(* Logix 5000 project; controller reports 1756-L63 rev 20.11; software revision 20.04; part 24 of 52 *)

        [1606].log_data[4].valid := 1, [1606].log_data[5].valid := 1, [1606].log_data[6].valid := 1, [1606].log_data[7].valid := 1, [1606].log_data[8].valid := 1, [1606].log_data[9].valid := 1, [1606].log_data[10].valid := 1, [1606].log_data[11].valid := 1, [1606].log_data[12].valid := 1, [1606].log_data[13].valid := 1, [1606].log_data[14].valid := 1, [1606].log_data[15].valid := 1, [1606].log_data[16].valid := 1, [1606].log_data[17].valid := 1, [1606].log_data[18].valid := 1, [1606].log_data[19].valid := 1, [1606].time.Year := 2023, [1606].time.Month := 1, [1606].time.Day := 15, [1606].time.Hour := 6, [1606].time.Minute := 14, [1606].time.Second := 59, [1607].log_data[0].min := 1.0, [1607].log_data[0].max := 1.0, [1607].log_data[0].total := 300.0, [1607].log_data[0].time := 300.0, [1607].log_data[0].minminute := 15, [1607].log_data[0].maxminute := 15, [1607].log_data[0].valid := 1, [1607].log_data[1].valid := 1, [1607].log_data[2].valid := 1, [1607].log_data[3].valid := 1, [1607].log_data[4].valid := 1, [1607].log_data[5].valid := 1, [1607].log_data[6].valid := 1, [1607].log_data[7].valid := 1, [1607].log_data[8].valid := 1, [1607].log_data[9].valid := 1, [1607].log_data[10].valid := 1, [1607].log_data[11].valid := 1, [1607].log_data[12].valid := 1, [1607].log_data[13].valid := 1, [1607].log_data[14].valid := 1, [1607].log_data[15].valid := 1, [1607].log_data[16].valid := 1, [1607].log_data[17].valid := 1, [1607].log_data[18].valid := 1, [1607].log_data[19].valid := 1, [1607].time.Year := 2023, [1607].time.Month := 1, [1607].time.Day := 15, [1607].time.Hour := 6, [1607].time.Minute := 19, [1607].time.Second := 59, [1608].log_data[0].min := 1.0, [1608].log_data[0].max := 1.0, [1608].log_data[0].total := 300.0, [1608].log_data[0].time := 300.0, [1608].log_data[0].minminute := 20, [1608].log_data[0].maxminute := 20,
        [1608].log_data[0].valid := 1, [1608].log_data[1].valid := 1, [1608].log_data[2].valid := 1, [1608].log_data[3].valid := 1, [1608].log_data[4].valid := 1, [1608].log_data[5].valid := 1, [1608].log_data[6].valid := 1, [1608].log_data[7].valid := 1, [1608].log_data[8].valid := 1, [1608].log_data[9].valid := 1, [1608].log_data[10].valid := 1, [1608].log_data[11].valid := 1, [1608].log_data[12].valid := 1, [1608].log_data[13].valid := 1, [1608].log_data[14].valid := 1, [1608].log_data[15].valid := 1, [1608].log_data[16].valid := 1, [1608].log_data[17].valid := 1, [1608].log_data[18].valid := 1, [1608].log_data[19].valid := 1, [1608].time.Year := 2023, [1608].time.Month := 1, [1608].time.Day := 15, [1608].time.Hour := 6, [1608].time.Minute := 24, [1608].time.Second := 59, [1609].log_data[0].min := 1.0, [1609].log_data[0].max := 1.0, [1609].log_data[0].total := 300.0, [1609].log_data[0].time := 300.0, [1609].log_data[0].minminute := 25, [1609].log_data[0].maxminute := 25, [1609].log_data[0].valid := 1, [1609].log_data[1].valid := 1, [1609].log_data[2].valid := 1, [1609].log_data[3].valid := 1, [1609].log_data[4].valid := 1, [1609].log_data[5].valid := 1, [1609].log_data[6].valid := 1, [1609].log_data[7].valid := 1, [1609].log_data[8].valid := 1, [1609].log_data[9].valid := 1, [1609].log_data[10].valid := 1, [1609].log_data[11].valid := 1, [1609].log_data[12].valid := 1, [1609].log_data[13].valid := 1, [1609].log_data[14].valid := 1, [1609].log_data[15].valid := 1, [1609].log_data[16].valid := 1, [1609].log_data[17].valid := 1, [1609].log_data[18].valid := 1, [1609].log_data[19].valid := 1, [1609].time.Year := 2023, [1609].time.Month := 1, [1609].time.Day := 15, [1609].time.Hour := 6, [1609].time.Minute := 29, [1609].time.Second := 59, [1610].log_data[0].min := 1.0, [1610].log_data[0].max := 1.0,
        [1610].log_data[0].total := 300.0, [1610].log_data[0].time := 300.0, [1610].log_data[0].minminute := 30, [1610].log_data[0].maxminute := 30, [1610].log_data[0].valid := 1, [1610].log_data[1].valid := 1, [1610].log_data[2].valid := 1, [1610].log_data[3].valid := 1, [1610].log_data[4].valid := 1, [1610].log_data[5].valid := 1, [1610].log_data[6].valid := 1, [1610].log_data[7].valid := 1, [1610].log_data[8].valid := 1, [1610].log_data[9].valid := 1, [1610].log_data[10].valid := 1, [1610].log_data[11].valid := 1, [1610].log_data[12].valid := 1, [1610].log_data[13].valid := 1, [1610].log_data[14].valid := 1, [1610].log_data[15].valid := 1, [1610].log_data[16].valid := 1, [1610].log_data[17].valid := 1, [1610].log_data[18].valid := 1, [1610].log_data[19].valid := 1, [1610].time.Year := 2023, [1610].time.Month := 1, [1610].time.Day := 15, [1610].time.Hour := 6, [1610].time.Minute := 34, [1610].time.Second := 59, [1611].log_data[0].min := 1.0, [1611].log_data[0].max := 1.0, [1611].log_data[0].total := 300.0, [1611].log_data[0].time := 300.0, [1611].log_data[0].minminute := 35, [1611].log_data[0].maxminute := 35, [1611].log_data[0].valid := 1, [1611].log_data[1].valid := 1, [1611].log_data[2].valid := 1, [1611].log_data[3].valid := 1, [1611].log_data[4].valid := 1, [1611].log_data[5].valid := 1, [1611].log_data[6].valid := 1, [1611].log_data[7].valid := 1, [1611].log_data[8].valid := 1, [1611].log_data[9].valid := 1, [1611].log_data[10].valid := 1, [1611].log_data[11].valid := 1, [1611].log_data[12].valid := 1, [1611].log_data[13].valid := 1, [1611].log_data[14].valid := 1, [1611].log_data[15].valid := 1, [1611].log_data[16].valid := 1, [1611].log_data[17].valid := 1, [1611].log_data[18].valid := 1, [1611].log_data[19].valid := 1, [1611].time.Year := 2023, [1611].time.Month := 1, [1611].time.Day := 15, [1611].time.Hour := 6,
        [1611].time.Minute := 39, [1611].time.Second := 59, [1612].log_data[0].min := 1.0, [1612].log_data[0].max := 1.0, [1612].log_data[0].total := 300.0, [1612].log_data[0].time := 300.0, [1612].log_data[0].minminute := 40, [1612].log_data[0].maxminute := 40, [1612].log_data[0].valid := 1, [1612].log_data[1].valid := 1, [1612].log_data[2].valid := 1, [1612].log_data[3].valid := 1, [1612].log_data[4].valid := 1, [1612].log_data[5].valid := 1, [1612].log_data[6].valid := 1, [1612].log_data[7].valid := 1, [1612].log_data[8].valid := 1, [1612].log_data[9].valid := 1, [1612].log_data[10].valid := 1, [1612].log_data[11].valid := 1, [1612].log_data[12].valid := 1, [1612].log_data[13].valid := 1, [1612].log_data[14].valid := 1, [1612].log_data[15].valid := 1, [1612].log_data[16].valid := 1, [1612].log_data[17].valid := 1, [1612].log_data[18].valid := 1, [1612].log_data[19].valid := 1, [1612].time.Year := 2023, [1612].time.Month := 1, [1612].time.Day := 15, [1612].time.Hour := 6, [1612].time.Minute := 44, [1612].time.Second := 59, [1613].log_data[0].min := 1.0, [1613].log_data[0].max := 1.0, [1613].log_data[0].total := 300.0, [1613].log_data[0].time := 300.0, [1613].log_data[0].minminute := 45, [1613].log_data[0].maxminute := 45, [1613].log_data[0].valid := 1, [1613].log_data[1].valid := 1, [1613].log_data[2].valid := 1, [1613].log_data[3].valid := 1, [1613].log_data[4].valid := 1, [1613].log_data[5].valid := 1, [1613].log_data[6].valid := 1, [1613].log_data[7].valid := 1, [1613].log_data[8].valid := 1, [1613].log_data[9].valid := 1, [1613].log_data[10].valid := 1, [1613].log_data[11].valid := 1, [1613].log_data[12].valid := 1, [1613].log_data[13].valid := 1, [1613].log_data[14].valid := 1, [1613].log_data[15].valid := 1, [1613].log_data[16].valid := 1, [1613].log_data[17].valid := 1, [1613].log_data[18].valid := 1, [1613].log_data[19].valid := 1,
        [1613].time.Year := 2023, [1613].time.Month := 1, [1613].time.Day := 15, [1613].time.Hour := 6, [1613].time.Minute := 49, [1613].time.Second := 59, [1614].log_data[0].min := 1.0, [1614].log_data[0].max := 1.0, [1614].log_data[0].total := 300.0, [1614].log_data[0].time := 300.0, [1614].log_data[0].minminute := 50, [1614].log_data[0].maxminute := 50, [1614].log_data[0].valid := 1, [1614].log_data[1].valid := 1, [1614].log_data[2].valid := 1, [1614].log_data[3].valid := 1, [1614].log_data[4].valid := 1, [1614].log_data[5].valid := 1, [1614].log_data[6].valid := 1, [1614].log_data[7].valid := 1, [1614].log_data[8].valid := 1, [1614].log_data[9].valid := 1, [1614].log_data[10].valid := 1, [1614].log_data[11].valid := 1, [1614].log_data[12].valid := 1, [1614].log_data[13].valid := 1, [1614].log_data[14].valid := 1, [1614].log_data[15].valid := 1, [1614].log_data[16].valid := 1, [1614].log_data[17].valid := 1, [1614].log_data[18].valid := 1, [1614].log_data[19].valid := 1, [1614].time.Year := 2023, [1614].time.Month := 1, [1614].time.Day := 15, [1614].time.Hour := 6, [1614].time.Minute := 54, [1614].time.Second := 59, [1615].log_data[0].min := 1.0, [1615].log_data[0].max := 1.0, [1615].log_data[0].total := 300.0, [1615].log_data[0].time := 300.0, [1615].log_data[0].minminute := 55, [1615].log_data[0].maxminute := 55, [1615].log_data[0].valid := 1, [1615].log_data[1].valid := 1, [1615].log_data[2].valid := 1, [1615].log_data[3].valid := 1, [1615].log_data[4].valid := 1, [1615].log_data[5].valid := 1, [1615].log_data[6].valid := 1, [1615].log_data[7].valid := 1, [1615].log_data[8].valid := 1, [1615].log_data[9].valid := 1, [1615].log_data[10].valid := 1, [1615].log_data[11].valid := 1, [1615].log_data[12].valid := 1, [1615].log_data[13].valid := 1, [1615].log_data[14].valid := 1, [1615].log_data[15].valid := 1,
        [1615].log_data[16].valid := 1, [1615].log_data[17].valid := 1, [1615].log_data[18].valid := 1, [1615].log_data[19].valid := 1, [1615].time.Year := 2023, [1615].time.Month := 1, [1615].time.Day := 15, [1615].time.Hour := 6, [1615].time.Minute := 59, [1615].time.Second := 59, [1616].log_data[0].min := 1.0, [1616].log_data[0].max := 1.0, [1616].log_data[0].total := 300.0, [1616].log_data[0].time := 300.0, [1616].log_data[0].valid := 1, [1616].log_data[1].valid := 1, [1616].log_data[2].valid := 1, [1616].log_data[3].valid := 1, [1616].log_data[4].valid := 1, [1616].log_data[5].valid := 1, [1616].log_data[6].valid := 1, [1616].log_data[7].valid := 1, [1616].log_data[8].valid := 1, [1616].log_data[9].valid := 1, [1616].log_data[10].valid := 1, [1616].log_data[11].valid := 1, [1616].log_data[12].valid := 1, [1616].log_data[13].valid := 1, [1616].log_data[14].valid := 1, [1616].log_data[15].valid := 1, [1616].log_data[16].valid := 1, [1616].log_data[17].valid := 1, [1616].log_data[18].valid := 1, [1616].log_data[19].valid := 1, [1616].time.Year := 2023, [1616].time.Month := 1, [1616].time.Day := 15, [1616].time.Hour := 7, [1616].time.Minute := 4, [1616].time.Second := 59, [1617].log_data[0].min := 1.0, [1617].log_data[0].max := 1.0, [1617].log_data[0].total := 300.0, [1617].log_data[0].time := 300.0, [1617].log_data[0].minminute := 5, [1617].log_data[0].maxminute := 5, [1617].log_data[0].valid := 1, [1617].log_data[1].valid := 1, [1617].log_data[2].valid := 1, [1617].log_data[3].valid := 1, [1617].log_data[4].valid := 1, [1617].log_data[5].valid := 1, [1617].log_data[6].valid := 1, [1617].log_data[7].valid := 1, [1617].log_data[8].valid := 1, [1617].log_data[9].valid := 1, [1617].log_data[10].valid := 1, [1617].log_data[11].valid := 1, [1617].log_data[12].valid := 1, [1617].log_data[13].valid := 1,
        [1617].log_data[14].valid := 1, [1617].log_data[15].valid := 1, [1617].log_data[16].valid := 1, [1617].log_data[17].valid := 1, [1617].log_data[18].valid := 1, [1617].log_data[19].valid := 1, [1617].time.Year := 2023, [1617].time.Month := 1, [1617].time.Day := 15, [1617].time.Hour := 7, [1617].time.Minute := 9, [1617].time.Second := 59, [1618].log_data[0].min := 1.0, [1618].log_data[0].max := 1.0, [1618].log_data[0].total := 300.0, [1618].log_data[0].time := 300.0, [1618].log_data[0].minminute := 10, [1618].log_data[0].maxminute := 10, [1618].log_data[0].valid := 1, [1618].log_data[1].valid := 1, [1618].log_data[2].valid := 1, [1618].log_data[3].valid := 1, [1618].log_data[4].valid := 1, [1618].log_data[5].valid := 1, [1618].log_data[6].valid := 1, [1618].log_data[7].valid := 1, [1618].log_data[8].valid := 1, [1618].log_data[9].valid := 1, [1618].log_data[10].valid := 1, [1618].log_data[11].valid := 1, [1618].log_data[12].valid := 1, [1618].log_data[13].valid := 1, [1618].log_data[14].valid := 1, [1618].log_data[15].valid := 1, [1618].log_data[16].valid := 1, [1618].log_data[17].valid := 1, [1618].log_data[18].valid := 1, [1618].log_data[19].valid := 1, [1618].time.Year := 2023, [1618].time.Month := 1, [1618].time.Day := 15, [1618].time.Hour := 7, [1618].time.Minute := 14, [1618].time.Second := 59, [1619].log_data[0].min := 1.0, [1619].log_data[0].max := 1.0, [1619].log_data[0].total := 300.0, [1619].log_data[0].time := 300.0, [1619].log_data[0].minminute := 15, [1619].log_data[0].maxminute := 15, [1619].log_data[0].valid := 1, [1619].log_data[1].valid := 1, [1619].log_data[2].valid := 1, [1619].log_data[3].valid := 1, [1619].log_data[4].valid := 1, [1619].log_data[5].valid := 1, [1619].log_data[6].valid := 1, [1619].log_data[7].valid := 1, [1619].log_data[8].valid := 1, [1619].log_data[9].valid := 1,
        [1619].log_data[10].valid := 1, [1619].log_data[11].valid := 1, [1619].log_data[12].valid := 1, [1619].log_data[13].valid := 1, [1619].log_data[14].valid := 1, [1619].log_data[15].valid := 1, [1619].log_data[16].valid := 1, [1619].log_data[17].valid := 1, [1619].log_data[18].valid := 1, [1619].log_data[19].valid := 1, [1619].time.Year := 2023, [1619].time.Month := 1, [1619].time.Day := 15, [1619].time.Hour := 7, [1619].time.Minute := 19, [1619].time.Second := 59, [1620].log_data[0].min := 1.0, [1620].log_data[0].max := 1.0, [1620].log_data[0].total := 300.0, [1620].log_data[0].time := 300.0, [1620].log_data[0].minminute := 20, [1620].log_data[0].maxminute := 20, [1620].log_data[0].valid := 1, [1620].log_data[1].valid := 1, [1620].log_data[2].valid := 1, [1620].log_data[3].valid := 1, [1620].log_data[4].valid := 1, [1620].log_data[5].valid := 1, [1620].log_data[6].valid := 1, [1620].log_data[7].valid := 1, [1620].log_data[8].valid := 1, [1620].log_data[9].valid := 1, [1620].log_data[10].valid := 1, [1620].log_data[11].valid := 1, [1620].log_data[12].valid := 1, [1620].log_data[13].valid := 1, [1620].log_data[14].valid := 1, [1620].log_data[15].valid := 1, [1620].log_data[16].valid := 1, [1620].log_data[17].valid := 1, [1620].log_data[18].valid := 1, [1620].log_data[19].valid := 1, [1620].time.Year := 2023, [1620].time.Month := 1, [1620].time.Day := 15, [1620].time.Hour := 7, [1620].time.Minute := 24, [1620].time.Second := 59, [1621].log_data[0].min := 1.0, [1621].log_data[0].max := 1.0, [1621].log_data[0].total := 300.0, [1621].log_data[0].time := 300.0, [1621].log_data[0].minminute := 25, [1621].log_data[0].maxminute := 25, [1621].log_data[0].valid := 1, [1621].log_data[1].valid := 1, [1621].log_data[2].valid := 1, [1621].log_data[3].valid := 1, [1621].log_data[4].valid := 1, [1621].log_data[5].valid := 1,
        [1621].log_data[6].valid := 1, [1621].log_data[7].valid := 1, [1621].log_data[8].valid := 1, [1621].log_data[9].valid := 1, [1621].log_data[10].valid := 1, [1621].log_data[11].valid := 1, [1621].log_data[12].valid := 1, [1621].log_data[13].valid := 1, [1621].log_data[14].valid := 1, [1621].log_data[15].valid := 1, [1621].log_data[16].valid := 1, [1621].log_data[17].valid := 1, [1621].log_data[18].valid := 1, [1621].log_data[19].valid := 1, [1621].time.Year := 2023, [1621].time.Month := 1, [1621].time.Day := 15, [1621].time.Hour := 7, [1621].time.Minute := 29, [1621].time.Second := 59, [1622].log_data[0].min := 1.0, [1622].log_data[0].max := 1.0, [1622].log_data[0].total := 300.0, [1622].log_data[0].time := 300.0, [1622].log_data[0].minminute := 30, [1622].log_data[0].maxminute := 30, [1622].log_data[0].valid := 1, [1622].log_data[1].valid := 1, [1622].log_data[2].valid := 1, [1622].log_data[3].valid := 1, [1622].log_data[4].valid := 1, [1622].log_data[5].valid := 1, [1622].log_data[6].valid := 1, [1622].log_data[7].valid := 1, [1622].log_data[8].valid := 1, [1622].log_data[9].valid := 1, [1622].log_data[10].valid := 1, [1622].log_data[11].valid := 1, [1622].log_data[12].valid := 1, [1622].log_data[13].valid := 1, [1622].log_data[14].valid := 1, [1622].log_data[15].valid := 1, [1622].log_data[16].valid := 1, [1622].log_data[17].valid := 1, [1622].log_data[18].valid := 1, [1622].log_data[19].valid := 1, [1622].time.Year := 2023, [1622].time.Month := 1, [1622].time.Day := 15, [1622].time.Hour := 7, [1622].time.Minute := 34, [1622].time.Second := 59, [1623].log_data[0].min := 1.0, [1623].log_data[0].max := 1.0, [1623].log_data[0].total := 300.0, [1623].log_data[0].time := 300.0, [1623].log_data[0].minminute := 35, [1623].log_data[0].maxminute := 35, [1623].log_data[0].valid := 1, [1623].log_data[1].valid := 1,
        [1623].log_data[2].valid := 1, [1623].log_data[3].valid := 1, [1623].log_data[4].valid := 1, [1623].log_data[5].valid := 1, [1623].log_data[6].valid := 1, [1623].log_data[7].valid := 1, [1623].log_data[8].valid := 1, [1623].log_data[9].valid := 1, [1623].log_data[10].valid := 1, [1623].log_data[11].valid := 1, [1623].log_data[12].valid := 1, [1623].log_data[13].valid := 1, [1623].log_data[14].valid := 1, [1623].log_data[15].valid := 1, [1623].log_data[16].valid := 1, [1623].log_data[17].valid := 1, [1623].log_data[18].valid := 1, [1623].log_data[19].valid := 1, [1623].time.Year := 2023, [1623].time.Month := 1, [1623].time.Day := 15, [1623].time.Hour := 7, [1623].time.Minute := 39, [1623].time.Second := 59, [1624].log_data[0].min := 1.0, [1624].log_data[0].max := 1.0, [1624].log_data[0].total := 300.0, [1624].log_data[0].time := 300.0, [1624].log_data[0].minminute := 40, [1624].log_data[0].maxminute := 40, [1624].log_data[0].valid := 1, [1624].log_data[1].valid := 1, [1624].log_data[2].valid := 1, [1624].log_data[3].valid := 1, [1624].log_data[4].valid := 1, [1624].log_data[5].valid := 1, [1624].log_data[6].valid := 1, [1624].log_data[7].valid := 1, [1624].log_data[8].valid := 1, [1624].log_data[9].valid := 1, [1624].log_data[10].valid := 1, [1624].log_data[11].valid := 1, [1624].log_data[12].valid := 1, [1624].log_data[13].valid := 1, [1624].log_data[14].valid := 1, [1624].log_data[15].valid := 1, [1624].log_data[16].valid := 1, [1624].log_data[17].valid := 1, [1624].log_data[18].valid := 1, [1624].log_data[19].valid := 1, [1624].time.Year := 2023, [1624].time.Month := 1, [1624].time.Day := 15, [1624].time.Hour := 7, [1624].time.Minute := 44, [1624].time.Second := 59, [1625].log_data[0].min := 1.0, [1625].log_data[0].max := 1.0, [1625].log_data[0].total := 300.0, [1625].log_data[0].time := 300.0,
        [1625].log_data[0].minminute := 45, [1625].log_data[0].maxminute := 45, [1625].log_data[0].valid := 1, [1625].log_data[1].valid := 1, [1625].log_data[2].valid := 1, [1625].log_data[3].valid := 1, [1625].log_data[4].valid := 1, [1625].log_data[5].valid := 1, [1625].log_data[6].valid := 1, [1625].log_data[7].valid := 1, [1625].log_data[8].valid := 1, [1625].log_data[9].valid := 1, [1625].log_data[10].valid := 1, [1625].log_data[11].valid := 1, [1625].log_data[12].valid := 1, [1625].log_data[13].valid := 1, [1625].log_data[14].valid := 1, [1625].log_data[15].valid := 1, [1625].log_data[16].valid := 1, [1625].log_data[17].valid := 1, [1625].log_data[18].valid := 1, [1625].log_data[19].valid := 1, [1625].time.Year := 2023, [1625].time.Month := 1, [1625].time.Day := 15, [1625].time.Hour := 7, [1625].time.Minute := 49, [1625].time.Second := 59, [1626].log_data[0].min := 1.0, [1626].log_data[0].max := 1.0, [1626].log_data[0].total := 300.0, [1626].log_data[0].time := 300.0, [1626].log_data[0].minminute := 50, [1626].log_data[0].maxminute := 50, [1626].log_data[0].valid := 1, [1626].log_data[1].valid := 1, [1626].log_data[2].valid := 1, [1626].log_data[3].valid := 1, [1626].log_data[4].valid := 1, [1626].log_data[5].valid := 1, [1626].log_data[6].valid := 1, [1626].log_data[7].valid := 1, [1626].log_data[8].valid := 1, [1626].log_data[9].valid := 1, [1626].log_data[10].valid := 1, [1626].log_data[11].valid := 1, [1626].log_data[12].valid := 1, [1626].log_data[13].valid := 1, [1626].log_data[14].valid := 1, [1626].log_data[15].valid := 1, [1626].log_data[16].valid := 1, [1626].log_data[17].valid := 1, [1626].log_data[18].valid := 1, [1626].log_data[19].valid := 1, [1626].time.Year := 2023, [1626].time.Month := 1, [1626].time.Day := 15, [1626].time.Hour := 7, [1626].time.Minute := 54, [1626].time.Second := 59,
        [1627].log_data[0].min := 1.0, [1627].log_data[0].max := 1.0, [1627].log_data[0].total := 300.0, [1627].log_data[0].time := 300.0, [1627].log_data[0].minminute := 55, [1627].log_data[0].maxminute := 55, [1627].log_data[0].valid := 1, [1627].log_data[1].valid := 1, [1627].log_data[2].valid := 1, [1627].log_data[3].valid := 1, [1627].log_data[4].valid := 1, [1627].log_data[5].valid := 1, [1627].log_data[6].valid := 1, [1627].log_data[7].valid := 1, [1627].log_data[8].valid := 1, [1627].log_data[9].valid := 1, [1627].log_data[10].valid := 1, [1627].log_data[11].valid := 1, [1627].log_data[12].valid := 1, [1627].log_data[13].valid := 1, [1627].log_data[14].valid := 1, [1627].log_data[15].valid := 1, [1627].log_data[16].valid := 1, [1627].log_data[17].valid := 1, [1627].log_data[18].valid := 1, [1627].log_data[19].valid := 1, [1627].time.Year := 2023, [1627].time.Month := 1, [1627].time.Day := 15, [1627].time.Hour := 7, [1627].time.Minute := 59, [1627].time.Second := 59, [1628].log_data[0].min := 1.0, [1628].log_data[0].max := 1.0, [1628].log_data[0].total := 300.0, [1628].log_data[0].time := 300.0, [1628].log_data[0].valid := 1, [1628].log_data[1].valid := 1, [1628].log_data[2].valid := 1, [1628].log_data[3].valid := 1, [1628].log_data[4].valid := 1, [1628].log_data[5].valid := 1, [1628].log_data[6].valid := 1, [1628].log_data[7].valid := 1, [1628].log_data[8].valid := 1, [1628].log_data[9].valid := 1, [1628].log_data[10].valid := 1, [1628].log_data[11].valid := 1, [1628].log_data[12].valid := 1, [1628].log_data[13].valid := 1, [1628].log_data[14].valid := 1, [1628].log_data[15].valid := 1, [1628].log_data[16].valid := 1, [1628].log_data[17].valid := 1, [1628].log_data[18].valid := 1, [1628].log_data[19].valid := 1, [1628].time.Year := 2023, [1628].time.Month := 1, [1628].time.Day := 15, [1628].time.Hour := 8,
        [1628].time.Minute := 4, [1628].time.Second := 59, [1629].log_data[0].min := 1.0, [1629].log_data[0].max := 1.0, [1629].log_data[0].total := 300.0, [1629].log_data[0].time := 300.0, [1629].log_data[0].minminute := 5, [1629].log_data[0].maxminute := 5, [1629].log_data[0].valid := 1, [1629].log_data[1].valid := 1, [1629].log_data[2].valid := 1, [1629].log_data[3].valid := 1, [1629].log_data[4].valid := 1, [1629].log_data[5].valid := 1, [1629].log_data[6].valid := 1, [1629].log_data[7].valid := 1, [1629].log_data[8].valid := 1, [1629].log_data[9].valid := 1, [1629].log_data[10].valid := 1, [1629].log_data[11].valid := 1, [1629].log_data[12].valid := 1, [1629].log_data[13].valid := 1, [1629].log_data[14].valid := 1, [1629].log_data[15].valid := 1, [1629].log_data[16].valid := 1, [1629].log_data[17].valid := 1, [1629].log_data[18].valid := 1, [1629].log_data[19].valid := 1, [1629].time.Year := 2023, [1629].time.Month := 1, [1629].time.Day := 15, [1629].time.Hour := 8, [1629].time.Minute := 9, [1629].time.Second := 59, [1630].log_data[0].min := 1.0, [1630].log_data[0].max := 1.0, [1630].log_data[0].total := 300.0, [1630].log_data[0].time := 300.0, [1630].log_data[0].minminute := 10, [1630].log_data[0].maxminute := 10, [1630].log_data[0].valid := 1, [1630].log_data[1].valid := 1, [1630].log_data[2].valid := 1, [1630].log_data[3].valid := 1, [1630].log_data[4].valid := 1, [1630].log_data[5].valid := 1, [1630].log_data[6].valid := 1, [1630].log_data[7].valid := 1, [1630].log_data[8].valid := 1, [1630].log_data[9].valid := 1, [1630].log_data[10].valid := 1, [1630].log_data[11].valid := 1, [1630].log_data[12].valid := 1, [1630].log_data[13].valid := 1, [1630].log_data[14].valid := 1, [1630].log_data[15].valid := 1, [1630].log_data[16].valid := 1, [1630].log_data[17].valid := 1, [1630].log_data[18].valid := 1, [1630].log_data[19].valid := 1,
        [1630].time.Year := 2023, [1630].time.Month := 1, [1630].time.Day := 15, [1630].time.Hour := 8, [1630].time.Minute := 14, [1630].time.Second := 59, [1631].log_data[0].min := 1.0, [1631].log_data[0].max := 1.0, [1631].log_data[0].total := 300.0, [1631].log_data[0].time := 300.0, [1631].log_data[0].minminute := 15, [1631].log_data[0].maxminute := 15, [1631].log_data[0].valid := 1, [1631].log_data[1].valid := 1, [1631].log_data[2].valid := 1, [1631].log_data[3].valid := 1, [1631].log_data[4].valid := 1, [1631].log_data[5].valid := 1, [1631].log_data[6].valid := 1, [1631].log_data[7].valid := 1, [1631].log_data[8].valid := 1, [1631].log_data[9].valid := 1, [1631].log_data[10].valid := 1, [1631].log_data[11].valid := 1, [1631].log_data[12].valid := 1, [1631].log_data[13].valid := 1, [1631].log_data[14].valid := 1, [1631].log_data[15].valid := 1, [1631].log_data[16].valid := 1, [1631].log_data[17].valid := 1, [1631].log_data[18].valid := 1, [1631].log_data[19].valid := 1, [1631].time.Year := 2023, [1631].time.Month := 1, [1631].time.Day := 15, [1631].time.Hour := 8, [1631].time.Minute := 19, [1631].time.Second := 59, [1632].log_data[0].min := 1.0, [1632].log_data[0].max := 1.0, [1632].log_data[0].total := 300.0, [1632].log_data[0].time := 300.0, [1632].log_data[0].minminute := 20, [1632].log_data[0].maxminute := 20, [1632].log_data[0].valid := 1, [1632].log_data[1].valid := 1, [1632].log_data[2].valid := 1, [1632].log_data[3].valid := 1, [1632].log_data[4].valid := 1, [1632].log_data[5].valid := 1, [1632].log_data[6].valid := 1, [1632].log_data[7].valid := 1, [1632].log_data[8].valid := 1, [1632].log_data[9].valid := 1, [1632].log_data[10].valid := 1, [1632].log_data[11].valid := 1, [1632].log_data[12].valid := 1, [1632].log_data[13].valid := 1, [1632].log_data[14].valid := 1, [1632].log_data[15].valid := 1,
        [1632].log_data[16].valid := 1, [1632].log_data[17].valid := 1, [1632].log_data[18].valid := 1, [1632].log_data[19].valid := 1, [1632].time.Year := 2023, [1632].time.Month := 1, [1632].time.Day := 15, [1632].time.Hour := 8, [1632].time.Minute := 24, [1632].time.Second := 59, [1633].log_data[0].min := 1.0, [1633].log_data[0].max := 1.0, [1633].log_data[0].total := 300.0, [1633].log_data[0].time := 300.0, [1633].log_data[0].minminute := 25, [1633].log_data[0].maxminute := 25, [1633].log_data[0].valid := 1, [1633].log_data[1].valid := 1, [1633].log_data[2].valid := 1, [1633].log_data[3].valid := 1, [1633].log_data[4].valid := 1, [1633].log_data[5].valid := 1, [1633].log_data[6].valid := 1, [1633].log_data[7].valid := 1, [1633].log_data[8].valid := 1, [1633].log_data[9].valid := 1, [1633].log_data[10].valid := 1, [1633].log_data[11].valid := 1, [1633].log_data[12].valid := 1, [1633].log_data[13].valid := 1, [1633].log_data[14].valid := 1, [1633].log_data[15].valid := 1, [1633].log_data[16].valid := 1, [1633].log_data[17].valid := 1, [1633].log_data[18].valid := 1, [1633].log_data[19].valid := 1, [1633].time.Year := 2023, [1633].time.Month := 1, [1633].time.Day := 15, [1633].time.Hour := 8, [1633].time.Minute := 29, [1633].time.Second := 59, [1634].log_data[0].min := 1.0, [1634].log_data[0].max := 1.0, [1634].log_data[0].total := 300.0, [1634].log_data[0].time := 300.0, [1634].log_data[0].minminute := 30, [1634].log_data[0].maxminute := 30, [1634].log_data[0].valid := 1, [1634].log_data[1].valid := 1, [1634].log_data[2].valid := 1, [1634].log_data[3].valid := 1, [1634].log_data[4].valid := 1, [1634].log_data[5].valid := 1, [1634].log_data[6].valid := 1, [1634].log_data[7].valid := 1, [1634].log_data[8].valid := 1, [1634].log_data[9].valid := 1, [1634].log_data[10].valid := 1, [1634].log_data[11].valid := 1,
        [1634].log_data[12].valid := 1, [1634].log_data[13].valid := 1, [1634].log_data[14].valid := 1, [1634].log_data[15].valid := 1, [1634].log_data[16].valid := 1, [1634].log_data[17].valid := 1, [1634].log_data[18].valid := 1, [1634].log_data[19].valid := 1, [1634].time.Year := 2023, [1634].time.Month := 1, [1634].time.Day := 15, [1634].time.Hour := 8, [1634].time.Minute := 34, [1634].time.Second := 59, [1635].log_data[0].min := 1.0, [1635].log_data[0].max := 1.0, [1635].log_data[0].total := 300.0, [1635].log_data[0].time := 300.0, [1635].log_data[0].minminute := 35, [1635].log_data[0].maxminute := 35, [1635].log_data[0].valid := 1, [1635].log_data[1].valid := 1, [1635].log_data[2].valid := 1, [1635].log_data[3].valid := 1, [1635].log_data[4].valid := 1, [1635].log_data[5].valid := 1, [1635].log_data[6].valid := 1, [1635].log_data[7].valid := 1, [1635].log_data[8].valid := 1, [1635].log_data[9].valid := 1, [1635].log_data[10].valid := 1, [1635].log_data[11].valid := 1, [1635].log_data[12].valid := 1, [1635].log_data[13].valid := 1, [1635].log_data[14].valid := 1, [1635].log_data[15].valid := 1, [1635].log_data[16].valid := 1, [1635].log_data[17].valid := 1, [1635].log_data[18].valid := 1, [1635].log_data[19].valid := 1, [1635].time.Year := 2023, [1635].time.Month := 1, [1635].time.Day := 15, [1635].time.Hour := 8, [1635].time.Minute := 39, [1635].time.Second := 59, [1636].log_data[0].min := 1.0, [1636].log_data[0].max := 1.0, [1636].log_data[0].total := 300.0, [1636].log_data[0].time := 300.0, [1636].log_data[0].minminute := 40, [1636].log_data[0].maxminute := 40, [1636].log_data[0].valid := 1, [1636].log_data[1].valid := 1, [1636].log_data[2].valid := 1, [1636].log_data[3].valid := 1, [1636].log_data[4].valid := 1, [1636].log_data[5].valid := 1, [1636].log_data[6].valid := 1, [1636].log_data[7].valid := 1,
        [1636].log_data[8].valid := 1, [1636].log_data[9].valid := 1, [1636].log_data[10].valid := 1, [1636].log_data[11].valid := 1, [1636].log_data[12].valid := 1, [1636].log_data[13].valid := 1, [1636].log_data[14].valid := 1, [1636].log_data[15].valid := 1, [1636].log_data[16].valid := 1, [1636].log_data[17].valid := 1, [1636].log_data[18].valid := 1, [1636].log_data[19].valid := 1, [1636].time.Year := 2023, [1636].time.Month := 1, [1636].time.Day := 15, [1636].time.Hour := 8, [1636].time.Minute := 44, [1636].time.Second := 59, [1637].log_data[0].min := 1.0, [1637].log_data[0].max := 1.0, [1637].log_data[0].total := 300.0, [1637].log_data[0].time := 300.0, [1637].log_data[0].minminute := 45, [1637].log_data[0].maxminute := 45, [1637].log_data[0].valid := 1, [1637].log_data[1].valid := 1, [1637].log_data[2].valid := 1, [1637].log_data[3].valid := 1, [1637].log_data[4].valid := 1, [1637].log_data[5].valid := 1, [1637].log_data[6].valid := 1, [1637].log_data[7].valid := 1, [1637].log_data[8].valid := 1, [1637].log_data[9].valid := 1, [1637].log_data[10].valid := 1, [1637].log_data[11].valid := 1, [1637].log_data[12].valid := 1, [1637].log_data[13].valid := 1, [1637].log_data[14].valid := 1, [1637].log_data[15].valid := 1, [1637].log_data[16].valid := 1, [1637].log_data[17].valid := 1, [1637].log_data[18].valid := 1, [1637].log_data[19].valid := 1, [1637].time.Year := 2023, [1637].time.Month := 1, [1637].time.Day := 15, [1637].time.Hour := 8, [1637].time.Minute := 49, [1637].time.Second := 59, [1638].log_data[0].min := 1.0, [1638].log_data[0].max := 1.0, [1638].log_data[0].total := 300.0, [1638].log_data[0].time := 300.0, [1638].log_data[0].minminute := 50, [1638].log_data[0].maxminute := 50, [1638].log_data[0].valid := 1, [1638].log_data[1].valid := 1, [1638].log_data[2].valid := 1, [1638].log_data[3].valid := 1,
        [1638].log_data[4].valid := 1, [1638].log_data[5].valid := 1, [1638].log_data[6].valid := 1, [1638].log_data[7].valid := 1, [1638].log_data[8].valid := 1, [1638].log_data[9].valid := 1, [1638].log_data[10].valid := 1, [1638].log_data[11].valid := 1, [1638].log_data[12].valid := 1, [1638].log_data[13].valid := 1, [1638].log_data[14].valid := 1, [1638].log_data[15].valid := 1, [1638].log_data[16].valid := 1, [1638].log_data[17].valid := 1, [1638].log_data[18].valid := 1, [1638].log_data[19].valid := 1, [1638].time.Year := 2023, [1638].time.Month := 1, [1638].time.Day := 15, [1638].time.Hour := 8, [1638].time.Minute := 54, [1638].time.Second := 59, [1639].log_data[0].min := 1.0, [1639].log_data[0].max := 1.0, [1639].log_data[0].total := 300.0, [1639].log_data[0].time := 300.0, [1639].log_data[0].minminute := 55, [1639].log_data[0].maxminute := 55, [1639].log_data[0].valid := 1, [1639].log_data[1].valid := 1, [1639].log_data[2].valid := 1, [1639].log_data[3].valid := 1, [1639].log_data[4].valid := 1, [1639].log_data[5].valid := 1, [1639].log_data[6].valid := 1, [1639].log_data[7].valid := 1, [1639].log_data[8].valid := 1, [1639].log_data[9].valid := 1, [1639].log_data[10].valid := 1, [1639].log_data[11].valid := 1, [1639].log_data[12].valid := 1, [1639].log_data[13].valid := 1, [1639].log_data[14].valid := 1, [1639].log_data[15].valid := 1, [1639].log_data[16].valid := 1, [1639].log_data[17].valid := 1, [1639].log_data[18].valid := 1, [1639].log_data[19].valid := 1, [1639].time.Year := 2023, [1639].time.Month := 1, [1639].time.Day := 15, [1639].time.Hour := 8, [1639].time.Minute := 59, [1639].time.Second := 59, [1640].log_data[0].min := 1.0, [1640].log_data[0].max := 1.0, [1640].log_data[0].total := 300.0, [1640].log_data[0].time := 300.0, [1640].log_data[0].valid := 1, [1640].log_data[1].valid := 1,
        [1640].log_data[2].valid := 1, [1640].log_data[3].valid := 1, [1640].log_data[4].valid := 1, [1640].log_data[5].valid := 1, [1640].log_data[6].valid := 1, [1640].log_data[7].valid := 1, [1640].log_data[8].valid := 1, [1640].log_data[9].valid := 1, [1640].log_data[10].valid := 1, [1640].log_data[11].valid := 1, [1640].log_data[12].valid := 1, [1640].log_data[13].valid := 1, [1640].log_data[14].valid := 1, [1640].log_data[15].valid := 1, [1640].log_data[16].valid := 1, [1640].log_data[17].valid := 1, [1640].log_data[18].valid := 1, [1640].log_data[19].valid := 1, [1640].time.Year := 2023, [1640].time.Month := 1, [1640].time.Day := 15, [1640].time.Hour := 9, [1640].time.Minute := 4, [1640].time.Second := 59, [1641].log_data[0].min := 1.0, [1641].log_data[0].max := 1.0, [1641].log_data[0].total := 300.0, [1641].log_data[0].time := 300.0, [1641].log_data[0].minminute := 5, [1641].log_data[0].maxminute := 5, [1641].log_data[0].valid := 1, [1641].log_data[1].valid := 1, [1641].log_data[2].valid := 1, [1641].log_data[3].valid := 1, [1641].log_data[4].valid := 1, [1641].log_data[5].valid := 1, [1641].log_data[6].valid := 1, [1641].log_data[7].valid := 1, [1641].log_data[8].valid := 1, [1641].log_data[9].valid := 1, [1641].log_data[10].valid := 1, [1641].log_data[11].valid := 1, [1641].log_data[12].valid := 1, [1641].log_data[13].valid := 1, [1641].log_data[14].valid := 1, [1641].log_data[15].valid := 1, [1641].log_data[16].valid := 1, [1641].log_data[17].valid := 1, [1641].log_data[18].valid := 1, [1641].log_data[19].valid := 1, [1641].time.Year := 2023, [1641].time.Month := 1, [1641].time.Day := 15, [1641].time.Hour := 9, [1641].time.Minute := 9, [1641].time.Second := 59, [1642].log_data[0].min := 1.0, [1642].log_data[0].max := 1.0, [1642].log_data[0].total := 300.0, [1642].log_data[0].time := 300.0,
        [1642].log_data[0].minminute := 10, [1642].log_data[0].maxminute := 10, [1642].log_data[0].valid := 1, [1642].log_data[1].valid := 1, [1642].log_data[2].valid := 1, [1642].log_data[3].valid := 1, [1642].log_data[4].valid := 1, [1642].log_data[5].valid := 1, [1642].log_data[6].valid := 1, [1642].log_data[7].valid := 1, [1642].log_data[8].valid := 1, [1642].log_data[9].valid := 1, [1642].log_data[10].valid := 1, [1642].log_data[11].valid := 1, [1642].log_data[12].valid := 1, [1642].log_data[13].valid := 1, [1642].log_data[14].valid := 1, [1642].log_data[15].valid := 1, [1642].log_data[16].valid := 1, [1642].log_data[17].valid := 1, [1642].log_data[18].valid := 1, [1642].log_data[19].valid := 1, [1642].time.Year := 2023, [1642].time.Month := 1, [1642].time.Day := 15, [1642].time.Hour := 9, [1642].time.Minute := 14, [1642].time.Second := 59, [1643].log_data[0].min := 1.0, [1643].log_data[0].max := 1.0, [1643].log_data[0].total := 300.0, [1643].log_data[0].time := 300.0, [1643].log_data[0].minminute := 15, [1643].log_data[0].maxminute := 15, [1643].log_data[0].valid := 1, [1643].log_data[1].valid := 1, [1643].log_data[2].valid := 1, [1643].log_data[3].valid := 1, [1643].log_data[4].valid := 1, [1643].log_data[5].valid := 1, [1643].log_data[6].valid := 1, [1643].log_data[7].valid := 1, [1643].log_data[8].valid := 1, [1643].log_data[9].valid := 1, [1643].log_data[10].valid := 1, [1643].log_data[11].valid := 1, [1643].log_data[12].valid := 1, [1643].log_data[13].valid := 1, [1643].log_data[14].valid := 1, [1643].log_data[15].valid := 1, [1643].log_data[16].valid := 1, [1643].log_data[17].valid := 1, [1643].log_data[18].valid := 1, [1643].log_data[19].valid := 1, [1643].time.Year := 2023, [1643].time.Month := 1, [1643].time.Day := 15, [1643].time.Hour := 9, [1643].time.Minute := 19, [1643].time.Second := 59,
        [1644].log_data[0].min := 1.0, [1644].log_data[0].max := 1.0, [1644].log_data[0].total := 300.0, [1644].log_data[0].time := 300.0, [1644].log_data[0].minminute := 20, [1644].log_data[0].maxminute := 20, [1644].log_data[0].valid := 1, [1644].log_data[1].valid := 1, [1644].log_data[2].valid := 1, [1644].log_data[3].valid := 1, [1644].log_data[4].valid := 1, [1644].log_data[5].valid := 1, [1644].log_data[6].valid := 1, [1644].log_data[7].valid := 1, [1644].log_data[8].valid := 1, [1644].log_data[9].valid := 1, [1644].log_data[10].valid := 1, [1644].log_data[11].valid := 1, [1644].log_data[12].valid := 1, [1644].log_data[13].valid := 1, [1644].log_data[14].valid := 1, [1644].log_data[15].valid := 1, [1644].log_data[16].valid := 1, [1644].log_data[17].valid := 1, [1644].log_data[18].valid := 1, [1644].log_data[19].valid := 1, [1644].time.Year := 2023, [1644].time.Month := 1, [1644].time.Day := 15, [1644].time.Hour := 9, [1644].time.Minute := 24, [1644].time.Second := 59, [1645].log_data[0].min := 1.0, [1645].log_data[0].max := 1.0, [1645].log_data[0].total := 300.0, [1645].log_data[0].time := 300.0, [1645].log_data[0].minminute := 25, [1645].log_data[0].maxminute := 25, [1645].log_data[0].valid := 1, [1645].log_data[1].valid := 1, [1645].log_data[2].valid := 1, [1645].log_data[3].valid := 1, [1645].log_data[4].valid := 1, [1645].log_data[5].valid := 1, [1645].log_data[6].valid := 1, [1645].log_data[7].valid := 1, [1645].log_data[8].valid := 1, [1645].log_data[9].valid := 1, [1645].log_data[10].valid := 1, [1645].log_data[11].valid := 1, [1645].log_data[12].valid := 1, [1645].log_data[13].valid := 1, [1645].log_data[14].valid := 1, [1645].log_data[15].valid := 1, [1645].log_data[16].valid := 1, [1645].log_data[17].valid := 1, [1645].log_data[18].valid := 1, [1645].log_data[19].valid := 1, [1645].time.Year := 2023, [1645].time.Month := 1,
        [1645].time.Day := 15, [1645].time.Hour := 9, [1645].time.Minute := 29, [1645].time.Second := 59, [1646].log_data[0].min := 1.0, [1646].log_data[0].max := 1.0, [1646].log_data[0].total := 300.0, [1646].log_data[0].time := 300.0, [1646].log_data[0].minminute := 30, [1646].log_data[0].maxminute := 30, [1646].log_data[0].valid := 1, [1646].log_data[1].valid := 1, [1646].log_data[2].valid := 1, [1646].log_data[3].valid := 1, [1646].log_data[4].valid := 1, [1646].log_data[5].valid := 1, [1646].log_data[6].valid := 1, [1646].log_data[7].valid := 1, [1646].log_data[8].valid := 1, [1646].log_data[9].valid := 1, [1646].log_data[10].valid := 1, [1646].log_data[11].valid := 1, [1646].log_data[12].valid := 1, [1646].log_data[13].valid := 1, [1646].log_data[14].valid := 1, [1646].log_data[15].valid := 1, [1646].log_data[16].valid := 1, [1646].log_data[17].valid := 1, [1646].log_data[18].valid := 1, [1646].log_data[19].valid := 1, [1646].time.Year := 2023, [1646].time.Month := 1, [1646].time.Day := 15, [1646].time.Hour := 9, [1646].time.Minute := 34, [1646].time.Second := 59, [1647].log_data[0].min := 1.0, [1647].log_data[0].max := 1.0, [1647].log_data[0].total := 300.0, [1647].log_data[0].time := 300.0, [1647].log_data[0].minminute := 35, [1647].log_data[0].maxminute := 35, [1647].log_data[0].valid := 1, [1647].log_data[1].valid := 1, [1647].log_data[2].valid := 1, [1647].log_data[3].valid := 1, [1647].log_data[4].valid := 1, [1647].log_data[5].valid := 1, [1647].log_data[6].valid := 1, [1647].log_data[7].valid := 1, [1647].log_data[8].valid := 1, [1647].log_data[9].valid := 1, [1647].log_data[10].valid := 1, [1647].log_data[11].valid := 1, [1647].log_data[12].valid := 1, [1647].log_data[13].valid := 1, [1647].log_data[14].valid := 1, [1647].log_data[15].valid := 1, [1647].log_data[16].valid := 1, [1647].log_data[17].valid := 1,
        [1647].log_data[18].valid := 1, [1647].log_data[19].valid := 1, [1647].time.Year := 2023, [1647].time.Month := 1, [1647].time.Day := 15, [1647].time.Hour := 9, [1647].time.Minute := 39, [1647].time.Second := 59, [1648].log_data[0].min := 1.0, [1648].log_data[0].max := 1.0, [1648].log_data[0].total := 300.0, [1648].log_data[0].time := 300.0, [1648].log_data[0].minminute := 40, [1648].log_data[0].maxminute := 40, [1648].log_data[0].valid := 1, [1648].log_data[1].valid := 1, [1648].log_data[2].valid := 1, [1648].log_data[3].valid := 1, [1648].log_data[4].valid := 1, [1648].log_data[5].valid := 1, [1648].log_data[6].valid := 1, [1648].log_data[7].valid := 1, [1648].log_data[8].valid := 1, [1648].log_data[9].valid := 1, [1648].log_data[10].valid := 1, [1648].log_data[11].valid := 1, [1648].log_data[12].valid := 1, [1648].log_data[13].valid := 1, [1648].log_data[14].valid := 1, [1648].log_data[15].valid := 1, [1648].log_data[16].valid := 1, [1648].log_data[17].valid := 1, [1648].log_data[18].valid := 1, [1648].log_data[19].valid := 1, [1648].time.Year := 2023, [1648].time.Month := 1, [1648].time.Day := 15, [1648].time.Hour := 9, [1648].time.Minute := 44, [1648].time.Second := 59, [1649].log_data[0].min := 1.0, [1649].log_data[0].max := 1.0, [1649].log_data[0].total := 300.0, [1649].log_data[0].time := 300.0, [1649].log_data[0].minminute := 45, [1649].log_data[0].maxminute := 45, [1649].log_data[0].valid := 1, [1649].log_data[1].valid := 1, [1649].log_data[2].valid := 1, [1649].log_data[3].valid := 1, [1649].log_data[4].valid := 1, [1649].log_data[5].valid := 1, [1649].log_data[6].valid := 1, [1649].log_data[7].valid := 1, [1649].log_data[8].valid := 1, [1649].log_data[9].valid := 1, [1649].log_data[10].valid := 1, [1649].log_data[11].valid := 1, [1649].log_data[12].valid := 1, [1649].log_data[13].valid := 1,
        [1649].log_data[14].valid := 1, [1649].log_data[15].valid := 1, [1649].log_data[16].valid := 1, [1649].log_data[17].valid := 1, [1649].log_data[18].valid := 1, [1649].log_data[19].valid := 1, [1649].time.Year := 2023, [1649].time.Month := 1, [1649].time.Day := 15, [1649].time.Hour := 9, [1649].time.Minute := 49, [1649].time.Second := 59, [1650].log_data[0].min := 1.0, [1650].log_data[0].max := 1.0, [1650].log_data[0].total := 300.0, [1650].log_data[0].time := 300.0, [1650].log_data[0].minminute := 50, [1650].log_data[0].maxminute := 50, [1650].log_data[0].valid := 1, [1650].log_data[1].valid := 1, [1650].log_data[2].valid := 1, [1650].log_data[3].valid := 1, [1650].log_data[4].valid := 1, [1650].log_data[5].valid := 1, [1650].log_data[6].valid := 1, [1650].log_data[7].valid := 1, [1650].log_data[8].valid := 1, [1650].log_data[9].valid := 1, [1650].log_data[10].valid := 1, [1650].log_data[11].valid := 1, [1650].log_data[12].valid := 1, [1650].log_data[13].valid := 1, [1650].log_data[14].valid := 1, [1650].log_data[15].valid := 1, [1650].log_data[16].valid := 1, [1650].log_data[17].valid := 1, [1650].log_data[18].valid := 1, [1650].log_data[19].valid := 1, [1650].time.Year := 2023, [1650].time.Month := 1, [1650].time.Day := 15, [1650].time.Hour := 9, [1650].time.Minute := 54, [1650].time.Second := 59, [1651].log_data[0].min := 1.0, [1651].log_data[0].max := 1.0, [1651].log_data[0].total := 300.0, [1651].log_data[0].time := 300.0, [1651].log_data[0].minminute := 55, [1651].log_data[0].maxminute := 55, [1651].log_data[0].valid := 1, [1651].log_data[1].valid := 1, [1651].log_data[2].valid := 1, [1651].log_data[3].valid := 1, [1651].log_data[4].valid := 1, [1651].log_data[5].valid := 1, [1651].log_data[6].valid := 1, [1651].log_data[7].valid := 1, [1651].log_data[8].valid := 1, [1651].log_data[9].valid := 1,
        [1651].log_data[10].valid := 1, [1651].log_data[11].valid := 1, [1651].log_data[12].valid := 1, [1651].log_data[13].valid := 1, [1651].log_data[14].valid := 1, [1651].log_data[15].valid := 1, [1651].log_data[16].valid := 1, [1651].log_data[17].valid := 1, [1651].log_data[18].valid := 1, [1651].log_data[19].valid := 1, [1651].time.Year := 2023, [1651].time.Month := 1, [1651].time.Day := 15, [1651].time.Hour := 9, [1651].time.Minute := 59, [1651].time.Second := 59, [1652].log_data[0].min := 1.0, [1652].log_data[0].max := 1.0, [1652].log_data[0].total := 300.0, [1652].log_data[0].time := 300.0, [1652].log_data[0].valid := 1, [1652].log_data[1].valid := 1, [1652].log_data[2].valid := 1, [1652].log_data[3].valid := 1, [1652].log_data[4].valid := 1, [1652].log_data[5].valid := 1, [1652].log_data[6].valid := 1, [1652].log_data[7].valid := 1, [1652].log_data[8].valid := 1, [1652].log_data[9].valid := 1, [1652].log_data[10].valid := 1, [1652].log_data[11].valid := 1, [1652].log_data[12].valid := 1, [1652].log_data[13].valid := 1, [1652].log_data[14].valid := 1, [1652].log_data[15].valid := 1, [1652].log_data[16].valid := 1, [1652].log_data[17].valid := 1, [1652].log_data[18].valid := 1, [1652].log_data[19].valid := 1, [1652].time.Year := 2023, [1652].time.Month := 1, [1652].time.Day := 15, [1652].time.Hour := 10, [1652].time.Minute := 4, [1652].time.Second := 59, [1653].log_data[0].min := 1.0, [1653].log_data[0].max := 1.0, [1653].log_data[0].total := 300.0, [1653].log_data[0].time := 300.0, [1653].log_data[0].minminute := 5, [1653].log_data[0].maxminute := 5, [1653].log_data[0].valid := 1, [1653].log_data[1].valid := 1, [1653].log_data[2].valid := 1, [1653].log_data[3].valid := 1, [1653].log_data[4].valid := 1, [1653].log_data[5].valid := 1, [1653].log_data[6].valid := 1, [1653].log_data[7].valid := 1,
        [1653].log_data[8].valid := 1, [1653].log_data[9].valid := 1, [1653].log_data[10].valid := 1, [1653].log_data[11].valid := 1, [1653].log_data[12].valid := 1, [1653].log_data[13].valid := 1, [1653].log_data[14].valid := 1, [1653].log_data[15].valid := 1, [1653].log_data[16].valid := 1, [1653].log_data[17].valid := 1, [1653].log_data[18].valid := 1, [1653].log_data[19].valid := 1, [1653].time.Year := 2023, [1653].time.Month := 1, [1653].time.Day := 15, [1653].time.Hour := 10, [1653].time.Minute := 9, [1653].time.Second := 59, [1654].log_data[0].min := 1.0, [1654].log_data[0].max := 1.0, [1654].log_data[0].total := 300.0, [1654].log_data[0].time := 300.0, [1654].log_data[0].minminute := 10, [1654].log_data[0].maxminute := 10, [1654].log_data[0].valid := 1, [1654].log_data[1].valid := 1, [1654].log_data[2].valid := 1, [1654].log_data[3].valid := 1, [1654].log_data[4].valid := 1, [1654].log_data[5].valid := 1, [1654].log_data[6].valid := 1, [1654].log_data[7].valid := 1, [1654].log_data[8].valid := 1, [1654].log_data[9].valid := 1, [1654].log_data[10].valid := 1, [1654].log_data[11].valid := 1, [1654].log_data[12].valid := 1, [1654].log_data[13].valid := 1, [1654].log_data[14].valid := 1, [1654].log_data[15].valid := 1, [1654].log_data[16].valid := 1, [1654].log_data[17].valid := 1, [1654].log_data[18].valid := 1, [1654].log_data[19].valid := 1, [1654].time.Year := 2023, [1654].time.Month := 1, [1654].time.Day := 15, [1654].time.Hour := 10, [1654].time.Minute := 14, [1654].time.Second := 59, [1655].log_data[0].min := 1.0, [1655].log_data[0].max := 1.0, [1655].log_data[0].total := 300.0, [1655].log_data[0].time := 300.0, [1655].log_data[0].minminute := 15, [1655].log_data[0].maxminute := 15, [1655].log_data[0].valid := 1, [1655].log_data[1].valid := 1, [1655].log_data[2].valid := 1, [1655].log_data[3].valid := 1,
        [1655].log_data[4].valid := 1, [1655].log_data[5].valid := 1, [1655].log_data[6].valid := 1, [1655].log_data[7].valid := 1, [1655].log_data[8].valid := 1, [1655].log_data[9].valid := 1, [1655].log_data[10].valid := 1, [1655].log_data[11].valid := 1, [1655].log_data[12].valid := 1, [1655].log_data[13].valid := 1, [1655].log_data[14].valid := 1, [1655].log_data[15].valid := 1, [1655].log_data[16].valid := 1, [1655].log_data[17].valid := 1, [1655].log_data[18].valid := 1, [1655].log_data[19].valid := 1, [1655].time.Year := 2023, [1655].time.Month := 1, [1655].time.Day := 15, [1655].time.Hour := 10, [1655].time.Minute := 19, [1655].time.Second := 59, [1656].log_data[0].min := 1.0, [1656].log_data[0].max := 1.0, [1656].log_data[0].total := 300.0, [1656].log_data[0].time := 300.0, [1656].log_data[0].minminute := 20, [1656].log_data[0].maxminute := 20, [1656].log_data[0].valid := 1, [1656].log_data[1].valid := 1, [1656].log_data[2].valid := 1, [1656].log_data[3].valid := 1, [1656].log_data[4].valid := 1, [1656].log_data[5].valid := 1, [1656].log_data[6].valid := 1, [1656].log_data[7].valid := 1, [1656].log_data[8].valid := 1, [1656].log_data[9].valid := 1, [1656].log_data[10].valid := 1, [1656].log_data[11].valid := 1, [1656].log_data[12].valid := 1, [1656].log_data[13].valid := 1, [1656].log_data[14].valid := 1, [1656].log_data[15].valid := 1, [1656].log_data[16].valid := 1, [1656].log_data[17].valid := 1, [1656].log_data[18].valid := 1, [1656].log_data[19].valid := 1, [1656].time.Year := 2023, [1656].time.Month := 1, [1656].time.Day := 15, [1656].time.Hour := 10, [1656].time.Minute := 24, [1656].time.Second := 59, [1657].log_data[0].min := 1.0, [1657].log_data[0].max := 1.0, [1657].log_data[0].total := 300.0, [1657].log_data[0].time := 300.0, [1657].log_data[0].minminute := 25, [1657].log_data[0].maxminute := 25,
        [1657].log_data[0].valid := 1, [1657].log_data[1].valid := 1, [1657].log_data[2].valid := 1, [1657].log_data[3].valid := 1, [1657].log_data[4].valid := 1, [1657].log_data[5].valid := 1, [1657].log_data[6].valid := 1, [1657].log_data[7].valid := 1, [1657].log_data[8].valid := 1, [1657].log_data[9].valid := 1, [1657].log_data[10].valid := 1, [1657].log_data[11].valid := 1, [1657].log_data[12].valid := 1, [1657].log_data[13].valid := 1, [1657].log_data[14].valid := 1, [1657].log_data[15].valid := 1, [1657].log_data[16].valid := 1, [1657].log_data[17].valid := 1, [1657].log_data[18].valid := 1, [1657].log_data[19].valid := 1, [1657].time.Year := 2023, [1657].time.Month := 1, [1657].time.Day := 15, [1657].time.Hour := 10, [1657].time.Minute := 29, [1657].time.Second := 59, [1658].log_data[0].min := 1.0, [1658].log_data[0].max := 1.0, [1658].log_data[0].total := 300.0, [1658].log_data[0].time := 300.0, [1658].log_data[0].minminute := 30, [1658].log_data[0].maxminute := 30, [1658].log_data[0].valid := 1, [1658].log_data[1].valid := 1, [1658].log_data[2].valid := 1, [1658].log_data[3].valid := 1, [1658].log_data[4].valid := 1, [1658].log_data[5].valid := 1, [1658].log_data[6].valid := 1, [1658].log_data[7].valid := 1, [1658].log_data[8].valid := 1, [1658].log_data[9].valid := 1, [1658].log_data[10].valid := 1, [1658].log_data[11].valid := 1, [1658].log_data[12].valid := 1, [1658].log_data[13].valid := 1, [1658].log_data[14].valid := 1, [1658].log_data[15].valid := 1, [1658].log_data[16].valid := 1, [1658].log_data[17].valid := 1, [1658].log_data[18].valid := 1, [1658].log_data[19].valid := 1, [1658].time.Year := 2023, [1658].time.Month := 1, [1658].time.Day := 15, [1658].time.Hour := 10, [1658].time.Minute := 34, [1658].time.Second := 59, [1659].log_data[0].min := 1.0, [1659].log_data[0].max := 1.0,
        [1659].log_data[0].total := 300.0, [1659].log_data[0].time := 300.0, [1659].log_data[0].minminute := 35, [1659].log_data[0].maxminute := 35, [1659].log_data[0].valid := 1, [1659].log_data[1].valid := 1, [1659].log_data[2].valid := 1, [1659].log_data[3].valid := 1, [1659].log_data[4].valid := 1, [1659].log_data[5].valid := 1, [1659].log_data[6].valid := 1, [1659].log_data[7].valid := 1, [1659].log_data[8].valid := 1, [1659].log_data[9].valid := 1, [1659].log_data[10].valid := 1, [1659].log_data[11].valid := 1, [1659].log_data[12].valid := 1, [1659].log_data[13].valid := 1, [1659].log_data[14].valid := 1, [1659].log_data[15].valid := 1, [1659].log_data[16].valid := 1, [1659].log_data[17].valid := 1, [1659].log_data[18].valid := 1, [1659].log_data[19].valid := 1, [1659].time.Year := 2023, [1659].time.Month := 1, [1659].time.Day := 15, [1659].time.Hour := 10, [1659].time.Minute := 39, [1659].time.Second := 59, [1660].log_data[0].min := 1.0, [1660].log_data[0].max := 1.0, [1660].log_data[0].total := 300.0, [1660].log_data[0].time := 300.0, [1660].log_data[0].minminute := 40, [1660].log_data[0].maxminute := 40, [1660].log_data[0].valid := 1, [1660].log_data[1].valid := 1, [1660].log_data[2].valid := 1, [1660].log_data[3].valid := 1, [1660].log_data[4].valid := 1, [1660].log_data[5].valid := 1, [1660].log_data[6].valid := 1, [1660].log_data[7].valid := 1, [1660].log_data[8].valid := 1, [1660].log_data[9].valid := 1, [1660].log_data[10].valid := 1, [1660].log_data[11].valid := 1, [1660].log_data[12].valid := 1, [1660].log_data[13].valid := 1, [1660].log_data[14].valid := 1, [1660].log_data[15].valid := 1, [1660].log_data[16].valid := 1, [1660].log_data[17].valid := 1, [1660].log_data[18].valid := 1, [1660].log_data[19].valid := 1, [1660].time.Year := 2023, [1660].time.Month := 1, [1660].time.Day := 15, [1660].time.Hour := 10,
        [1660].time.Minute := 44, [1660].time.Second := 59, [1661].log_data[0].min := 1.0, [1661].log_data[0].max := 1.0, [1661].log_data[0].total := 300.0, [1661].log_data[0].time := 300.0, [1661].log_data[0].minminute := 45, [1661].log_data[0].maxminute := 45, [1661].log_data[0].valid := 1, [1661].log_data[1].valid := 1, [1661].log_data[2].valid := 1, [1661].log_data[3].valid := 1, [1661].log_data[4].valid := 1, [1661].log_data[5].valid := 1, [1661].log_data[6].valid := 1, [1661].log_data[7].valid := 1, [1661].log_data[8].valid := 1, [1661].log_data[9].valid := 1, [1661].log_data[10].valid := 1, [1661].log_data[11].valid := 1, [1661].log_data[12].valid := 1, [1661].log_data[13].valid := 1, [1661].log_data[14].valid := 1, [1661].log_data[15].valid := 1, [1661].log_data[16].valid := 1, [1661].log_data[17].valid := 1, [1661].log_data[18].valid := 1, [1661].log_data[19].valid := 1, [1661].time.Year := 2023, [1661].time.Month := 1, [1661].time.Day := 15, [1661].time.Hour := 10, [1661].time.Minute := 49, [1661].time.Second := 59, [1662].log_data[0].min := 1.0, [1662].log_data[0].max := 1.0, [1662].log_data[0].total := 300.0, [1662].log_data[0].time := 300.0, [1662].log_data[0].minminute := 50, [1662].log_data[0].maxminute := 50, [1662].log_data[0].valid := 1, [1662].log_data[1].valid := 1, [1662].log_data[2].valid := 1, [1662].log_data[3].valid := 1, [1662].log_data[4].valid := 1, [1662].log_data[5].valid := 1, [1662].log_data[6].valid := 1, [1662].log_data[7].valid := 1, [1662].log_data[8].valid := 1, [1662].log_data[9].valid := 1, [1662].log_data[10].valid := 1, [1662].log_data[11].valid := 1, [1662].log_data[12].valid := 1, [1662].log_data[13].valid := 1, [1662].log_data[14].valid := 1, [1662].log_data[15].valid := 1, [1662].log_data[16].valid := 1, [1662].log_data[17].valid := 1, [1662].log_data[18].valid := 1, [1662].log_data[19].valid := 1,
        [1662].time.Year := 2023, [1662].time.Month := 1, [1662].time.Day := 15, [1662].time.Hour := 10, [1662].time.Minute := 54, [1662].time.Second := 59, [1663].log_data[0].min := 1.0, [1663].log_data[0].max := 1.0, [1663].log_data[0].total := 300.0, [1663].log_data[0].time := 300.0, [1663].log_data[0].minminute := 55, [1663].log_data[0].maxminute := 55, [1663].log_data[0].valid := 1, [1663].log_data[1].valid := 1, [1663].log_data[2].valid := 1, [1663].log_data[3].valid := 1, [1663].log_data[4].valid := 1, [1663].log_data[5].valid := 1, [1663].log_data[6].valid := 1, [1663].log_data[7].valid := 1, [1663].log_data[8].valid := 1, [1663].log_data[9].valid := 1, [1663].log_data[10].valid := 1, [1663].log_data[11].valid := 1, [1663].log_data[12].valid := 1, [1663].log_data[13].valid := 1, [1663].log_data[14].valid := 1, [1663].log_data[15].valid := 1, [1663].log_data[16].valid := 1, [1663].log_data[17].valid := 1, [1663].log_data[18].valid := 1, [1663].log_data[19].valid := 1, [1663].time.Year := 2023, [1663].time.Month := 1, [1663].time.Day := 15, [1663].time.Hour := 10, [1663].time.Minute := 59, [1663].time.Second := 59, [1664].log_data[0].min := 1.0, [1664].log_data[0].max := 1.0, [1664].log_data[0].total := 299.5, [1664].log_data[0].time := 299.5, [1664].log_data[0].valid := 1, [1664].log_data[1].valid := 1, [1664].log_data[2].valid := 1, [1664].log_data[3].valid := 1, [1664].log_data[4].valid := 1, [1664].log_data[5].valid := 1, [1664].log_data[6].valid := 1, [1664].log_data[7].valid := 1, [1664].log_data[8].valid := 1, [1664].log_data[9].valid := 1, [1664].log_data[10].valid := 1, [1664].log_data[11].valid := 1, [1664].log_data[12].valid := 1, [1664].log_data[13].valid := 1, [1664].log_data[14].valid := 1, [1664].log_data[15].valid := 1, [1664].log_data[16].valid := 1, [1664].log_data[17].valid := 1,
        [1664].log_data[18].valid := 1, [1664].log_data[19].valid := 1, [1664].time.Year := 2023, [1664].time.Month := 1, [1664].time.Day := 15, [1664].time.Hour := 11, [1664].time.Minute := 4, [1664].time.Second := 59, [1665].log_data[0].min := 1.0, [1665].log_data[0].max := 1.0, [1665].log_data[0].total := 300.0, [1665].log_data[0].time := 300.0, [1665].log_data[0].minminute := 5, [1665].log_data[0].maxminute := 5, [1665].log_data[0].valid := 1, [1665].log_data[1].valid := 1, [1665].log_data[2].valid := 1, [1665].log_data[3].valid := 1, [1665].log_data[4].valid := 1, [1665].log_data[5].valid := 1, [1665].log_data[6].valid := 1, [1665].log_data[7].valid := 1, [1665].log_data[8].valid := 1, [1665].log_data[9].valid := 1, [1665].log_data[10].valid := 1, [1665].log_data[11].valid := 1, [1665].log_data[12].valid := 1, [1665].log_data[13].valid := 1, [1665].log_data[14].valid := 1, [1665].log_data[15].valid := 1, [1665].log_data[16].valid := 1, [1665].log_data[17].valid := 1, [1665].log_data[18].valid := 1, [1665].log_data[19].valid := 1, [1665].time.Year := 2023, [1665].time.Month := 1, [1665].time.Day := 15, [1665].time.Hour := 11, [1665].time.Minute := 9, [1665].time.Second := 59, [1666].log_data[0].min := 1.0, [1666].log_data[0].max := 1.0, [1666].log_data[0].total := 300.0, [1666].log_data[0].time := 300.0, [1666].log_data[0].minminute := 10, [1666].log_data[0].maxminute := 10, [1666].log_data[0].valid := 1, [1666].log_data[1].valid := 1, [1666].log_data[2].valid := 1, [1666].log_data[3].valid := 1, [1666].log_data[4].valid := 1, [1666].log_data[5].valid := 1, [1666].log_data[6].valid := 1, [1666].log_data[7].valid := 1, [1666].log_data[8].valid := 1, [1666].log_data[9].valid := 1, [1666].log_data[10].valid := 1, [1666].log_data[11].valid := 1, [1666].log_data[12].valid := 1, [1666].log_data[13].valid := 1,
        [1666].log_data[14].valid := 1, [1666].log_data[15].valid := 1, [1666].log_data[16].valid := 1, [1666].log_data[17].valid := 1, [1666].log_data[18].valid := 1, [1666].log_data[19].valid := 1, [1666].time.Year := 2023, [1666].time.Month := 1, [1666].time.Day := 15, [1666].time.Hour := 11, [1666].time.Minute := 14, [1666].time.Second := 59, [1667].log_data[0].min := 1.0, [1667].log_data[0].max := 1.0, [1667].log_data[0].total := 300.0, [1667].log_data[0].time := 300.0, [1667].log_data[0].minminute := 15, [1667].log_data[0].maxminute := 15, [1667].log_data[0].valid := 1, [1667].log_data[1].valid := 1, [1667].log_data[2].valid := 1, [1667].log_data[3].valid := 1, [1667].log_data[4].valid := 1, [1667].log_data[5].valid := 1, [1667].log_data[6].valid := 1, [1667].log_data[7].valid := 1, [1667].log_data[8].valid := 1, [1667].log_data[9].valid := 1, [1667].log_data[10].valid := 1, [1667].log_data[11].valid := 1, [1667].log_data[12].valid := 1, [1667].log_data[13].valid := 1, [1667].log_data[14].valid := 1, [1667].log_data[15].valid := 1, [1667].log_data[16].valid := 1, [1667].log_data[17].valid := 1, [1667].log_data[18].valid := 1, [1667].log_data[19].valid := 1, [1667].time.Year := 2023, [1667].time.Month := 1, [1667].time.Day := 15, [1667].time.Hour := 11, [1667].time.Minute := 19, [1667].time.Second := 59, [1668].log_data[0].min := 1.0, [1668].log_data[0].max := 1.0, [1668].log_data[0].total := 300.0, [1668].log_data[0].time := 300.0, [1668].log_data[0].minminute := 20, [1668].log_data[0].maxminute := 20, [1668].log_data[0].valid := 1, [1668].log_data[1].valid := 1, [1668].log_data[2].valid := 1, [1668].log_data[3].valid := 1, [1668].log_data[4].valid := 1, [1668].log_data[5].valid := 1, [1668].log_data[6].valid := 1, [1668].log_data[7].valid := 1, [1668].log_data[8].valid := 1, [1668].log_data[9].valid := 1,
        [1668].log_data[10].valid := 1, [1668].log_data[11].valid := 1, [1668].log_data[12].valid := 1, [1668].log_data[13].valid := 1, [1668].log_data[14].valid := 1, [1668].log_data[15].valid := 1, [1668].log_data[16].valid := 1, [1668].log_data[17].valid := 1, [1668].log_data[18].valid := 1, [1668].log_data[19].valid := 1, [1668].time.Year := 2023, [1668].time.Month := 1, [1668].time.Day := 15, [1668].time.Hour := 11, [1668].time.Minute := 24, [1668].time.Second := 59, [1669].log_data[0].min := 1.0, [1669].log_data[0].max := 1.0, [1669].log_data[0].total := 300.0, [1669].log_data[0].time := 300.0, [1669].log_data[0].minminute := 25, [1669].log_data[0].maxminute := 25, [1669].log_data[0].valid := 1, [1669].log_data[1].valid := 1, [1669].log_data[2].valid := 1, [1669].log_data[3].valid := 1, [1669].log_data[4].valid := 1, [1669].log_data[5].valid := 1, [1669].log_data[6].valid := 1, [1669].log_data[7].valid := 1, [1669].log_data[8].valid := 1, [1669].log_data[9].valid := 1, [1669].log_data[10].valid := 1, [1669].log_data[11].valid := 1, [1669].log_data[12].valid := 1, [1669].log_data[13].valid := 1, [1669].log_data[14].valid := 1, [1669].log_data[15].valid := 1, [1669].log_data[16].valid := 1, [1669].log_data[17].valid := 1, [1669].log_data[18].valid := 1, [1669].log_data[19].valid := 1, [1669].time.Year := 2023, [1669].time.Month := 1, [1669].time.Day := 15, [1669].time.Hour := 11, [1669].time.Minute := 29, [1669].time.Second := 59, [1670].log_data[0].min := 1.0, [1670].log_data[0].max := 1.0, [1670].log_data[0].total := 300.0, [1670].log_data[0].time := 300.0, [1670].log_data[0].minminute := 30, [1670].log_data[0].maxminute := 30, [1670].log_data[0].valid := 1, [1670].log_data[1].valid := 1, [1670].log_data[2].valid := 1, [1670].log_data[3].valid := 1, [1670].log_data[4].valid := 1, [1670].log_data[5].valid := 1,
        [1670].log_data[6].valid := 1, [1670].log_data[7].valid := 1, [1670].log_data[8].valid := 1, [1670].log_data[9].valid := 1, [1670].log_data[10].valid := 1, [1670].log_data[11].valid := 1, [1670].log_data[12].valid := 1, [1670].log_data[13].valid := 1, [1670].log_data[14].valid := 1, [1670].log_data[15].valid := 1, [1670].log_data[16].valid := 1, [1670].log_data[17].valid := 1, [1670].log_data[18].valid := 1, [1670].log_data[19].valid := 1, [1670].time.Year := 2023, [1670].time.Month := 1, [1670].time.Day := 15, [1670].time.Hour := 11, [1670].time.Minute := 34, [1670].time.Second := 59, [1671].log_data[0].min := 1.0, [1671].log_data[0].max := 1.0, [1671].log_data[0].total := 300.0, [1671].log_data[0].time := 300.0, [1671].log_data[0].minminute := 35, [1671].log_data[0].maxminute := 35, [1671].log_data[0].valid := 1, [1671].log_data[1].valid := 1, [1671].log_data[2].valid := 1, [1671].log_data[3].valid := 1, [1671].log_data[4].valid := 1, [1671].log_data[5].valid := 1, [1671].log_data[6].valid := 1, [1671].log_data[7].valid := 1, [1671].log_data[8].valid := 1, [1671].log_data[9].valid := 1, [1671].log_data[10].valid := 1, [1671].log_data[11].valid := 1, [1671].log_data[12].valid := 1, [1671].log_data[13].valid := 1, [1671].log_data[14].valid := 1, [1671].log_data[15].valid := 1, [1671].log_data[16].valid := 1, [1671].log_data[17].valid := 1, [1671].log_data[18].valid := 1, [1671].log_data[19].valid := 1, [1671].time.Year := 2023, [1671].time.Month := 1, [1671].time.Day := 15, [1671].time.Hour := 11, [1671].time.Minute := 39, [1671].time.Second := 59, [1672].log_data[0].min := 1.0, [1672].log_data[0].max := 1.0, [1672].log_data[0].total := 300.0, [1672].log_data[0].time := 300.0, [1672].log_data[0].minminute := 40, [1672].log_data[0].maxminute := 40, [1672].log_data[0].valid := 1, [1672].log_data[1].valid := 1,
        [1672].log_data[2].valid := 1, [1672].log_data[3].valid := 1, [1672].log_data[4].valid := 1, [1672].log_data[5].valid := 1, [1672].log_data[6].valid := 1, [1672].log_data[7].valid := 1, [1672].log_data[8].valid := 1, [1672].log_data[9].valid := 1, [1672].log_data[10].valid := 1, [1672].log_data[11].valid := 1, [1672].log_data[12].valid := 1, [1672].log_data[13].valid := 1, [1672].log_data[14].valid := 1, [1672].log_data[15].valid := 1, [1672].log_data[16].valid := 1, [1672].log_data[17].valid := 1, [1672].log_data[18].valid := 1, [1672].log_data[19].valid := 1, [1672].time.Year := 2023, [1672].time.Month := 1, [1672].time.Day := 15, [1672].time.Hour := 11, [1672].time.Minute := 44, [1672].time.Second := 59, [1673].log_data[0].min := 1.0, [1673].log_data[0].max := 1.0, [1673].log_data[0].total := 300.0, [1673].log_data[0].time := 300.0, [1673].log_data[0].minminute := 45, [1673].log_data[0].maxminute := 45, [1673].log_data[0].valid := 1, [1673].log_data[1].valid := 1, [1673].log_data[2].valid := 1, [1673].log_data[3].valid := 1, [1673].log_data[4].valid := 1, [1673].log_data[5].valid := 1, [1673].log_data[6].valid := 1, [1673].log_data[7].valid := 1, [1673].log_data[8].valid := 1, [1673].log_data[9].valid := 1, [1673].log_data[10].valid := 1, [1673].log_data[11].valid := 1, [1673].log_data[12].valid := 1, [1673].log_data[13].valid := 1, [1673].log_data[14].valid := 1, [1673].log_data[15].valid := 1, [1673].log_data[16].valid := 1, [1673].log_data[17].valid := 1, [1673].log_data[18].valid := 1, [1673].log_data[19].valid := 1, [1673].time.Year := 2023, [1673].time.Month := 1, [1673].time.Day := 15, [1673].time.Hour := 11, [1673].time.Minute := 49, [1673].time.Second := 59, [1674].log_data[0].min := 1.0, [1674].log_data[0].max := 1.0, [1674].log_data[0].total := 300.0, [1674].log_data[0].time := 300.0,
        [1674].log_data[0].minminute := 50, [1674].log_data[0].maxminute := 50, [1674].log_data[0].valid := 1, [1674].log_data[1].valid := 1, [1674].log_data[2].valid := 1, [1674].log_data[3].valid := 1, [1674].log_data[4].valid := 1, [1674].log_data[5].valid := 1, [1674].log_data[6].valid := 1, [1674].log_data[7].valid := 1, [1674].log_data[8].valid := 1, [1674].log_data[9].valid := 1, [1674].log_data[10].valid := 1, [1674].log_data[11].valid := 1, [1674].log_data[12].valid := 1, [1674].log_data[13].valid := 1, [1674].log_data[14].valid := 1, [1674].log_data[15].valid := 1, [1674].log_data[16].valid := 1, [1674].log_data[17].valid := 1, [1674].log_data[18].valid := 1, [1674].log_data[19].valid := 1, [1674].time.Year := 2023, [1674].time.Month := 1, [1674].time.Day := 15, [1674].time.Hour := 11, [1674].time.Minute := 54, [1674].time.Second := 59, [1675].log_data[0].min := 1.0, [1675].log_data[0].max := 1.0, [1675].log_data[0].total := 300.0, [1675].log_data[0].time := 300.0, [1675].log_data[0].minminute := 55, [1675].log_data[0].maxminute := 55, [1675].log_data[0].valid := 1, [1675].log_data[1].valid := 1, [1675].log_data[2].valid := 1, [1675].log_data[3].valid := 1, [1675].log_data[4].valid := 1, [1675].log_data[5].valid := 1, [1675].log_data[6].valid := 1, [1675].log_data[7].valid := 1, [1675].log_data[8].valid := 1, [1675].log_data[9].valid := 1, [1675].log_data[10].valid := 1, [1675].log_data[11].valid := 1, [1675].log_data[12].valid := 1, [1675].log_data[13].valid := 1, [1675].log_data[14].valid := 1, [1675].log_data[15].valid := 1, [1675].log_data[16].valid := 1, [1675].log_data[17].valid := 1, [1675].log_data[18].valid := 1, [1675].log_data[19].valid := 1, [1675].time.Year := 2023, [1675].time.Month := 1, [1675].time.Day := 15, [1675].time.Hour := 11, [1675].time.Minute := 59, [1675].time.Second := 59,
        [1676].log_data[0].min := 1.0, [1676].log_data[0].max := 1.0, [1676].log_data[0].total := 300.0, [1676].log_data[0].time := 300.0, [1676].log_data[0].valid := 1, [1676].log_data[1].valid := 1, [1676].log_data[2].valid := 1, [1676].log_data[3].valid := 1, [1676].log_data[4].valid := 1, [1676].log_data[5].valid := 1, [1676].log_data[6].valid := 1, [1676].log_data[7].valid := 1, [1676].log_data[8].valid := 1, [1676].log_data[9].valid := 1, [1676].log_data[10].valid := 1, [1676].log_data[11].valid := 1, [1676].log_data[12].valid := 1, [1676].log_data[13].valid := 1, [1676].log_data[14].valid := 1, [1676].log_data[15].valid := 1, [1676].log_data[16].valid := 1, [1676].log_data[17].valid := 1, [1676].log_data[18].valid := 1, [1676].log_data[19].valid := 1, [1676].time.Year := 2023, [1676].time.Month := 1, [1676].time.Day := 15, [1676].time.Hour := 12, [1676].time.Minute := 4, [1676].time.Second := 59, [1677].log_data[0].min := 1.0, [1677].log_data[0].max := 1.0, [1677].log_data[0].total := 300.0, [1677].log_data[0].time := 300.0, [1677].log_data[0].minminute := 5, [1677].log_data[0].maxminute := 5, [1677].log_data[0].valid := 1, [1677].log_data[1].valid := 1, [1677].log_data[2].valid := 1, [1677].log_data[3].valid := 1, [1677].log_data[4].valid := 1, [1677].log_data[5].valid := 1, [1677].log_data[6].valid := 1, [1677].log_data[7].valid := 1, [1677].log_data[8].valid := 1, [1677].log_data[9].valid := 1, [1677].log_data[10].valid := 1, [1677].log_data[11].valid := 1, [1677].log_data[12].valid := 1, [1677].log_data[13].valid := 1, [1677].log_data[14].valid := 1, [1677].log_data[15].valid := 1, [1677].log_data[16].valid := 1, [1677].log_data[17].valid := 1, [1677].log_data[18].valid := 1, [1677].log_data[19].valid := 1, [1677].time.Year := 2023, [1677].time.Month := 1, [1677].time.Day := 15, [1677].time.Hour := 12,
        [1677].time.Minute := 9, [1677].time.Second := 59, [1678].log_data[0].min := 1.0, [1678].log_data[0].max := 1.0, [1678].log_data[0].total := 300.0, [1678].log_data[0].time := 300.0, [1678].log_data[0].minminute := 10, [1678].log_data[0].maxminute := 10, [1678].log_data[0].valid := 1, [1678].log_data[1].valid := 1, [1678].log_data[2].valid := 1, [1678].log_data[3].valid := 1, [1678].log_data[4].valid := 1, [1678].log_data[5].valid := 1, [1678].log_data[6].valid := 1, [1678].log_data[7].valid := 1, [1678].log_data[8].valid := 1, [1678].log_data[9].valid := 1, [1678].log_data[10].valid := 1, [1678].log_data[11].valid := 1, [1678].log_data[12].valid := 1, [1678].log_data[13].valid := 1, [1678].log_data[14].valid := 1, [1678].log_data[15].valid := 1, [1678].log_data[16].valid := 1, [1678].log_data[17].valid := 1, [1678].log_data[18].valid := 1, [1678].log_data[19].valid := 1, [1678].time.Year := 2023, [1678].time.Month := 1, [1678].time.Day := 15, [1678].time.Hour := 12, [1678].time.Minute := 14, [1678].time.Second := 59, [1679].log_data[0].min := 1.0, [1679].log_data[0].max := 1.0, [1679].log_data[0].total := 300.0, [1679].log_data[0].time := 300.0, [1679].log_data[0].minminute := 15, [1679].log_data[0].maxminute := 15, [1679].log_data[0].valid := 1, [1679].log_data[1].valid := 1, [1679].log_data[2].valid := 1, [1679].log_data[3].valid := 1, [1679].log_data[4].valid := 1, [1679].log_data[5].valid := 1, [1679].log_data[6].valid := 1, [1679].log_data[7].valid := 1, [1679].log_data[8].valid := 1, [1679].log_data[9].valid := 1, [1679].log_data[10].valid := 1, [1679].log_data[11].valid := 1, [1679].log_data[12].valid := 1, [1679].log_data[13].valid := 1, [1679].log_data[14].valid := 1, [1679].log_data[15].valid := 1, [1679].log_data[16].valid := 1, [1679].log_data[17].valid := 1, [1679].log_data[18].valid := 1, [1679].log_data[19].valid := 1,
        [1679].time.Year := 2023, [1679].time.Month := 1, [1679].time.Day := 15, [1679].time.Hour := 12, [1679].time.Minute := 19, [1679].time.Second := 59, [1680].log_data[0].min := 1.0, [1680].log_data[0].max := 1.0, [1680].log_data[0].total := 300.0, [1680].log_data[0].time := 300.0, [1680].log_data[0].minminute := 20, [1680].log_data[0].maxminute := 20, [1680].log_data[0].valid := 1, [1680].log_data[1].valid := 1, [1680].log_data[2].valid := 1, [1680].log_data[3].valid := 1, [1680].log_data[4].valid := 1, [1680].log_data[5].valid := 1, [1680].log_data[6].valid := 1, [1680].log_data[7].valid := 1, [1680].log_data[8].valid := 1, [1680].log_data[9].valid := 1, [1680].log_data[10].valid := 1, [1680].log_data[11].valid := 1, [1680].log_data[12].valid := 1, [1680].log_data[13].valid := 1, [1680].log_data[14].valid := 1, [1680].log_data[15].valid := 1, [1680].log_data[16].valid := 1, [1680].log_data[17].valid := 1, [1680].log_data[18].valid := 1, [1680].log_data[19].valid := 1, [1680].time.Year := 2023, [1680].time.Month := 1, [1680].time.Day := 15, [1680].time.Hour := 12, [1680].time.Minute := 24, [1680].time.Second := 59, [1681].log_data[0].min := 1.0, [1681].log_data[0].max := 1.0, [1681].log_data[0].total := 300.0, [1681].log_data[0].time := 300.0, [1681].log_data[0].minminute := 25, [1681].log_data[0].maxminute := 25, [1681].log_data[0].valid := 1, [1681].log_data[1].valid := 1, [1681].log_data[2].valid := 1, [1681].log_data[3].valid := 1, [1681].log_data[4].valid := 1, [1681].log_data[5].valid := 1, [1681].log_data[6].valid := 1, [1681].log_data[7].valid := 1, [1681].log_data[8].valid := 1, [1681].log_data[9].valid := 1, [1681].log_data[10].valid := 1, [1681].log_data[11].valid := 1, [1681].log_data[12].valid := 1, [1681].log_data[13].valid := 1, [1681].log_data[14].valid := 1, [1681].log_data[15].valid := 1,
        [1681].log_data[16].valid := 1, [1681].log_data[17].valid := 1, [1681].log_data[18].valid := 1, [1681].log_data[19].valid := 1, [1681].time.Year := 2023, [1681].time.Month := 1, [1681].time.Day := 15, [1681].time.Hour := 12, [1681].time.Minute := 29, [1681].time.Second := 59, [1682].log_data[0].min := 1.0, [1682].log_data[0].max := 1.0, [1682].log_data[0].total := 300.0, [1682].log_data[0].time := 300.0, [1682].log_data[0].minminute := 30, [1682].log_data[0].maxminute := 30, [1682].log_data[0].valid := 1, [1682].log_data[1].valid := 1, [1682].log_data[2].valid := 1, [1682].log_data[3].valid := 1, [1682].log_data[4].valid := 1, [1682].log_data[5].valid := 1, [1682].log_data[6].valid := 1, [1682].log_data[7].valid := 1, [1682].log_data[8].valid := 1, [1682].log_data[9].valid := 1, [1682].log_data[10].valid := 1, [1682].log_data[11].valid := 1, [1682].log_data[12].valid := 1, [1682].log_data[13].valid := 1, [1682].log_data[14].valid := 1, [1682].log_data[15].valid := 1, [1682].log_data[16].valid := 1, [1682].log_data[17].valid := 1, [1682].log_data[18].valid := 1, [1682].log_data[19].valid := 1, [1682].time.Year := 2023, [1682].time.Month := 1, [1682].time.Day := 15, [1682].time.Hour := 12, [1682].time.Minute := 34, [1682].time.Second := 59, [1683].log_data[0].min := 1.0, [1683].log_data[0].max := 1.0, [1683].log_data[0].total := 300.0, [1683].log_data[0].time := 300.0, [1683].log_data[0].minminute := 35, [1683].log_data[0].maxminute := 35, [1683].log_data[0].valid := 1, [1683].log_data[1].valid := 1, [1683].log_data[2].valid := 1, [1683].log_data[3].valid := 1, [1683].log_data[4].valid := 1, [1683].log_data[5].valid := 1, [1683].log_data[6].valid := 1, [1683].log_data[7].valid := 1, [1683].log_data[8].valid := 1, [1683].log_data[9].valid := 1, [1683].log_data[10].valid := 1, [1683].log_data[11].valid := 1,
        [1683].log_data[12].valid := 1, [1683].log_data[13].valid := 1, [1683].log_data[14].valid := 1, [1683].log_data[15].valid := 1, [1683].log_data[16].valid := 1, [1683].log_data[17].valid := 1, [1683].log_data[18].valid := 1, [1683].log_data[19].valid := 1, [1683].time.Year := 2023, [1683].time.Month := 1, [1683].time.Day := 15, [1683].time.Hour := 12, [1683].time.Minute := 39, [1683].time.Second := 59, [1684].log_data[0].min := 1.0, [1684].log_data[0].max := 1.0, [1684].log_data[0].total := 300.0, [1684].log_data[0].time := 300.0, [1684].log_data[0].minminute := 40, [1684].log_data[0].maxminute := 40, [1684].log_data[0].valid := 1, [1684].log_data[1].valid := 1, [1684].log_data[2].valid := 1, [1684].log_data[3].valid := 1, [1684].log_data[4].valid := 1, [1684].log_data[5].valid := 1, [1684].log_data[6].valid := 1, [1684].log_data[7].valid := 1, [1684].log_data[8].valid := 1, [1684].log_data[9].valid := 1, [1684].log_data[10].valid := 1, [1684].log_data[11].valid := 1, [1684].log_data[12].valid := 1, [1684].log_data[13].valid := 1, [1684].log_data[14].valid := 1, [1684].log_data[15].valid := 1, [1684].log_data[16].valid := 1, [1684].log_data[17].valid := 1, [1684].log_data[18].valid := 1, [1684].log_data[19].valid := 1, [1684].time.Year := 2023, [1684].time.Month := 1, [1684].time.Day := 15, [1684].time.Hour := 12, [1684].time.Minute := 44, [1684].time.Second := 59, [1685].log_data[0].min := 1.0, [1685].log_data[0].max := 1.0, [1685].log_data[0].total := 300.0, [1685].log_data[0].time := 300.0, [1685].log_data[0].minminute := 45, [1685].log_data[0].maxminute := 45, [1685].log_data[0].valid := 1, [1685].log_data[1].valid := 1, [1685].log_data[2].valid := 1, [1685].log_data[3].valid := 1, [1685].log_data[4].valid := 1, [1685].log_data[5].valid := 1, [1685].log_data[6].valid := 1, [1685].log_data[7].valid := 1,
        [1685].log_data[8].valid := 1, [1685].log_data[9].valid := 1, [1685].log_data[10].valid := 1, [1685].log_data[11].valid := 1, [1685].log_data[12].valid := 1, [1685].log_data[13].valid := 1, [1685].log_data[14].valid := 1, [1685].log_data[15].valid := 1, [1685].log_data[16].valid := 1, [1685].log_data[17].valid := 1, [1685].log_data[18].valid := 1, [1685].log_data[19].valid := 1, [1685].time.Year := 2023, [1685].time.Month := 1, [1685].time.Day := 15, [1685].time.Hour := 12, [1685].time.Minute := 49, [1685].time.Second := 59, [1686].log_data[0].min := 1.0, [1686].log_data[0].max := 1.0, [1686].log_data[0].total := 300.0, [1686].log_data[0].time := 300.0, [1686].log_data[0].minminute := 50, [1686].log_data[0].maxminute := 50, [1686].log_data[0].valid := 1, [1686].log_data[1].valid := 1, [1686].log_data[2].valid := 1, [1686].log_data[3].valid := 1, [1686].log_data[4].valid := 1, [1686].log_data[5].valid := 1, [1686].log_data[6].valid := 1, [1686].log_data[7].valid := 1, [1686].log_data[8].valid := 1, [1686].log_data[9].valid := 1, [1686].log_data[10].valid := 1, [1686].log_data[11].valid := 1, [1686].log_data[12].valid := 1, [1686].log_data[13].valid := 1, [1686].log_data[14].valid := 1, [1686].log_data[15].valid := 1, [1686].log_data[16].valid := 1, [1686].log_data[17].valid := 1, [1686].log_data[18].valid := 1, [1686].log_data[19].valid := 1, [1686].time.Year := 2023, [1686].time.Month := 1, [1686].time.Day := 15, [1686].time.Hour := 12, [1686].time.Minute := 54, [1686].time.Second := 59, [1687].log_data[0].min := 1.0, [1687].log_data[0].max := 1.0, [1687].log_data[0].total := 300.0, [1687].log_data[0].time := 300.0, [1687].log_data[0].minminute := 55, [1687].log_data[0].maxminute := 55, [1687].log_data[0].valid := 1, [1687].log_data[1].valid := 1, [1687].log_data[2].valid := 1, [1687].log_data[3].valid := 1,
        [1687].log_data[4].valid := 1, [1687].log_data[5].valid := 1, [1687].log_data[6].valid := 1, [1687].log_data[7].valid := 1, [1687].log_data[8].valid := 1, [1687].log_data[9].valid := 1, [1687].log_data[10].valid := 1, [1687].log_data[11].valid := 1, [1687].log_data[12].valid := 1, [1687].log_data[13].valid := 1, [1687].log_data[14].valid := 1, [1687].log_data[15].valid := 1, [1687].log_data[16].valid := 1, [1687].log_data[17].valid := 1, [1687].log_data[18].valid := 1, [1687].log_data[19].valid := 1, [1687].time.Year := 2023, [1687].time.Month := 1, [1687].time.Day := 15, [1687].time.Hour := 12, [1687].time.Minute := 59, [1687].time.Second := 59, [1688].log_data[0].min := 1.0, [1688].log_data[0].max := 1.0, [1688].log_data[0].total := 300.0, [1688].log_data[0].time := 300.0, [1688].log_data[0].valid := 1, [1688].log_data[1].valid := 1, [1688].log_data[2].valid := 1, [1688].log_data[3].valid := 1, [1688].log_data[4].valid := 1, [1688].log_data[5].valid := 1, [1688].log_data[6].valid := 1, [1688].log_data[7].valid := 1, [1688].log_data[8].valid := 1, [1688].log_data[9].valid := 1, [1688].log_data[10].valid := 1, [1688].log_data[11].valid := 1, [1688].log_data[12].valid := 1, [1688].log_data[13].valid := 1, [1688].log_data[14].valid := 1, [1688].log_data[15].valid := 1, [1688].log_data[16].valid := 1, [1688].log_data[17].valid := 1, [1688].log_data[18].valid := 1, [1688].log_data[19].valid := 1, [1688].time.Year := 2023, [1688].time.Month := 1, [1688].time.Day := 15, [1688].time.Hour := 13, [1688].time.Minute := 4, [1688].time.Second := 59, [1689].log_data[0].min := 1.0, [1689].log_data[0].max := 1.0, [1689].log_data[0].total := 300.0, [1689].log_data[0].time := 300.0, [1689].log_data[0].minminute := 5, [1689].log_data[0].maxminute := 5, [1689].log_data[0].valid := 1, [1689].log_data[1].valid := 1,
        [1689].log_data[2].valid := 1, [1689].log_data[3].valid := 1, [1689].log_data[4].valid := 1, [1689].log_data[5].valid := 1, [1689].log_data[6].valid := 1, [1689].log_data[7].valid := 1, [1689].log_data[8].valid := 1, [1689].log_data[9].valid := 1, [1689].log_data[10].valid := 1, [1689].log_data[11].valid := 1, [1689].log_data[12].valid := 1, [1689].log_data[13].valid := 1, [1689].log_data[14].valid := 1, [1689].log_data[15].valid := 1, [1689].log_data[16].valid := 1, [1689].log_data[17].valid := 1, [1689].log_data[18].valid := 1, [1689].log_data[19].valid := 1, [1689].time.Year := 2023, [1689].time.Month := 1, [1689].time.Day := 15, [1689].time.Hour := 13, [1689].time.Minute := 9, [1689].time.Second := 59, [1690].log_data[0].min := 1.0, [1690].log_data[0].max := 1.0, [1690].log_data[0].total := 300.0, [1690].log_data[0].time := 300.0, [1690].log_data[0].minminute := 10, [1690].log_data[0].maxminute := 10, [1690].log_data[0].valid := 1, [1690].log_data[1].valid := 1, [1690].log_data[2].valid := 1, [1690].log_data[3].valid := 1, [1690].log_data[4].valid := 1, [1690].log_data[5].valid := 1, [1690].log_data[6].valid := 1, [1690].log_data[7].valid := 1, [1690].log_data[8].valid := 1, [1690].log_data[9].valid := 1, [1690].log_data[10].valid := 1, [1690].log_data[11].valid := 1, [1690].log_data[12].valid := 1, [1690].log_data[13].valid := 1, [1690].log_data[14].valid := 1, [1690].log_data[15].valid := 1, [1690].log_data[16].valid := 1, [1690].log_data[17].valid := 1, [1690].log_data[18].valid := 1, [1690].log_data[19].valid := 1, [1690].time.Year := 2023, [1690].time.Month := 1, [1690].time.Day := 15, [1690].time.Hour := 13, [1690].time.Minute := 14, [1690].time.Second := 59, [1691].log_data[0].min := 1.0, [1691].log_data[0].max := 1.0, [1691].log_data[0].total := 300.0, [1691].log_data[0].time := 300.0,
        [1691].log_data[0].minminute := 15, [1691].log_data[0].maxminute := 15, [1691].log_data[0].valid := 1, [1691].log_data[1].valid := 1, [1691].log_data[2].valid := 1, [1691].log_data[3].valid := 1, [1691].log_data[4].valid := 1, [1691].log_data[5].valid := 1, [1691].log_data[6].valid := 1, [1691].log_data[7].valid := 1, [1691].log_data[8].valid := 1, [1691].log_data[9].valid := 1, [1691].log_data[10].valid := 1, [1691].log_data[11].valid := 1, [1691].log_data[12].valid := 1, [1691].log_data[13].valid := 1, [1691].log_data[14].valid := 1, [1691].log_data[15].valid := 1, [1691].log_data[16].valid := 1, [1691].log_data[17].valid := 1, [1691].log_data[18].valid := 1, [1691].log_data[19].valid := 1, [1691].time.Year := 2023, [1691].time.Month := 1, [1691].time.Day := 15, [1691].time.Hour := 13, [1691].time.Minute := 19, [1691].time.Second := 59, [1692].log_data[0].min := 1.0, [1692].log_data[0].max := 1.0, [1692].log_data[0].total := 300.0, [1692].log_data[0].time := 300.0, [1692].log_data[0].minminute := 20, [1692].log_data[0].maxminute := 20, [1692].log_data[0].valid := 1, [1692].log_data[1].valid := 1, [1692].log_data[2].valid := 1, [1692].log_data[3].valid := 1, [1692].log_data[4].valid := 1, [1692].log_data[5].valid := 1, [1692].log_data[6].valid := 1, [1692].log_data[7].valid := 1, [1692].log_data[8].valid := 1, [1692].log_data[9].valid := 1, [1692].log_data[10].valid := 1, [1692].log_data[11].valid := 1, [1692].log_data[12].valid := 1, [1692].log_data[13].valid := 1, [1692].log_data[14].valid := 1, [1692].log_data[15].valid := 1, [1692].log_data[16].valid := 1, [1692].log_data[17].valid := 1, [1692].log_data[18].valid := 1, [1692].log_data[19].valid := 1, [1692].time.Year := 2023, [1692].time.Month := 1, [1692].time.Day := 15, [1692].time.Hour := 13, [1692].time.Minute := 24, [1692].time.Second := 59,
        [1693].log_data[0].min := 1.0, [1693].log_data[0].max := 1.0, [1693].log_data[0].total := 300.0, [1693].log_data[0].time := 300.0, [1693].log_data[0].minminute := 25, [1693].log_data[0].maxminute := 25, [1693].log_data[0].valid := 1, [1693].log_data[1].valid := 1, [1693].log_data[2].valid := 1, [1693].log_data[3].valid := 1, [1693].log_data[4].valid := 1, [1693].log_data[5].valid := 1, [1693].log_data[6].valid := 1, [1693].log_data[7].valid := 1, [1693].log_data[8].valid := 1, [1693].log_data[9].valid := 1, [1693].log_data[10].valid := 1, [1693].log_data[11].valid := 1, [1693].log_data[12].valid := 1, [1693].log_data[13].valid := 1, [1693].log_data[14].valid := 1, [1693].log_data[15].valid := 1, [1693].log_data[16].valid := 1, [1693].log_data[17].valid := 1, [1693].log_data[18].valid := 1, [1693].log_data[19].valid := 1, [1693].time.Year := 2023, [1693].time.Month := 1, [1693].time.Day := 15, [1693].time.Hour := 13, [1693].time.Minute := 29, [1693].time.Second := 59, [1694].log_data[0].min := 1.0, [1694].log_data[0].max := 1.0, [1694].log_data[0].total := 300.0, [1694].log_data[0].time := 300.0, [1694].log_data[0].minminute := 30, [1694].log_data[0].maxminute := 30, [1694].log_data[0].valid := 1, [1694].log_data[1].valid := 1, [1694].log_data[2].valid := 1, [1694].log_data[3].valid := 1, [1694].log_data[4].valid := 1, [1694].log_data[5].valid := 1, [1694].log_data[6].valid := 1, [1694].log_data[7].valid := 1, [1694].log_data[8].valid := 1, [1694].log_data[9].valid := 1, [1694].log_data[10].valid := 1, [1694].log_data[11].valid := 1, [1694].log_data[12].valid := 1, [1694].log_data[13].valid := 1, [1694].log_data[14].valid := 1, [1694].log_data[15].valid := 1, [1694].log_data[16].valid := 1, [1694].log_data[17].valid := 1, [1694].log_data[18].valid := 1, [1694].log_data[19].valid := 1, [1694].time.Year := 2023, [1694].time.Month := 1,
        [1694].time.Day := 15, [1694].time.Hour := 13, [1694].time.Minute := 34, [1694].time.Second := 59, [1695].log_data[0].min := 1.0, [1695].log_data[0].max := 1.0, [1695].log_data[0].total := 300.0, [1695].log_data[0].time := 300.0, [1695].log_data[0].minminute := 35, [1695].log_data[0].maxminute := 35, [1695].log_data[0].valid := 1, [1695].log_data[1].valid := 1, [1695].log_data[2].valid := 1, [1695].log_data[3].valid := 1, [1695].log_data[4].valid := 1, [1695].log_data[5].valid := 1, [1695].log_data[6].valid := 1, [1695].log_data[7].valid := 1, [1695].log_data[8].valid := 1, [1695].log_data[9].valid := 1, [1695].log_data[10].valid := 1, [1695].log_data[11].valid := 1, [1695].log_data[12].valid := 1, [1695].log_data[13].valid := 1, [1695].log_data[14].valid := 1, [1695].log_data[15].valid := 1, [1695].log_data[16].valid := 1, [1695].log_data[17].valid := 1, [1695].log_data[18].valid := 1, [1695].log_data[19].valid := 1, [1695].time.Year := 2023, [1695].time.Month := 1, [1695].time.Day := 15, [1695].time.Hour := 13, [1695].time.Minute := 39, [1695].time.Second := 59, [1696].log_data[0].min := 1.0, [1696].log_data[0].max := 1.0, [1696].log_data[0].total := 300.0, [1696].log_data[0].time := 300.0, [1696].log_data[0].minminute := 40, [1696].log_data[0].maxminute := 40, [1696].log_data[0].valid := 1, [1696].log_data[1].valid := 1, [1696].log_data[2].valid := 1, [1696].log_data[3].valid := 1, [1696].log_data[4].valid := 1, [1696].log_data[5].valid := 1, [1696].log_data[6].valid := 1, [1696].log_data[7].valid := 1, [1696].log_data[8].valid := 1, [1696].log_data[9].valid := 1, [1696].log_data[10].valid := 1, [1696].log_data[11].valid := 1, [1696].log_data[12].valid := 1, [1696].log_data[13].valid := 1, [1696].log_data[14].valid := 1, [1696].log_data[15].valid := 1, [1696].log_data[16].valid := 1, [1696].log_data[17].valid := 1,
        [1696].log_data[18].valid := 1, [1696].log_data[19].valid := 1, [1696].time.Year := 2023, [1696].time.Month := 1, [1696].time.Day := 15, [1696].time.Hour := 13, [1696].time.Minute := 44, [1696].time.Second := 59, [1697].log_data[0].min := 1.0, [1697].log_data[0].max := 1.0, [1697].log_data[0].total := 300.0, [1697].log_data[0].time := 300.0, [1697].log_data[0].minminute := 45, [1697].log_data[0].maxminute := 45, [1697].log_data[0].valid := 1, [1697].log_data[1].valid := 1, [1697].log_data[2].valid := 1, [1697].log_data[3].valid := 1, [1697].log_data[4].valid := 1, [1697].log_data[5].valid := 1, [1697].log_data[6].valid := 1, [1697].log_data[7].valid := 1, [1697].log_data[8].valid := 1, [1697].log_data[9].valid := 1, [1697].log_data[10].valid := 1, [1697].log_data[11].valid := 1, [1697].log_data[12].valid := 1, [1697].log_data[13].valid := 1, [1697].log_data[14].valid := 1, [1697].log_data[15].valid := 1, [1697].log_data[16].valid := 1, [1697].log_data[17].valid := 1, [1697].log_data[18].valid := 1, [1697].log_data[19].valid := 1, [1697].time.Year := 2023, [1697].time.Month := 1, [1697].time.Day := 15, [1697].time.Hour := 13, [1697].time.Minute := 49, [1697].time.Second := 59, [1698].log_data[0].min := 1.0, [1698].log_data[0].max := 1.0, [1698].log_data[0].total := 300.0, [1698].log_data[0].time := 300.0, [1698].log_data[0].minminute := 50, [1698].log_data[0].maxminute := 50, [1698].log_data[0].valid := 1, [1698].log_data[1].valid := 1, [1698].log_data[2].valid := 1, [1698].log_data[3].valid := 1, [1698].log_data[4].valid := 1, [1698].log_data[5].valid := 1, [1698].log_data[6].valid := 1, [1698].log_data[7].valid := 1, [1698].log_data[8].valid := 1, [1698].log_data[9].valid := 1, [1698].log_data[10].valid := 1, [1698].log_data[11].valid := 1, [1698].log_data[12].valid := 1, [1698].log_data[13].valid := 1,
        [1698].log_data[14].valid := 1, [1698].log_data[15].valid := 1, [1698].log_data[16].valid := 1, [1698].log_data[17].valid := 1, [1698].log_data[18].valid := 1, [1698].log_data[19].valid := 1, [1698].time.Year := 2023, [1698].time.Month := 1, [1698].time.Day := 15, [1698].time.Hour := 13, [1698].time.Minute := 54, [1698].time.Second := 59, [1699].log_data[0].min := 1.0, [1699].log_data[0].max := 1.0, [1699].log_data[0].total := 300.0, [1699].log_data[0].time := 300.0, [1699].log_data[0].minminute := 55, [1699].log_data[0].maxminute := 55, [1699].log_data[0].valid := 1, [1699].log_data[1].valid := 1, [1699].log_data[2].valid := 1, [1699].log_data[3].valid := 1, [1699].log_data[4].valid := 1, [1699].log_data[5].valid := 1, [1699].log_data[6].valid := 1, [1699].log_data[7].valid := 1, [1699].log_data[8].valid := 1, [1699].log_data[9].valid := 1, [1699].log_data[10].valid := 1, [1699].log_data[11].valid := 1, [1699].log_data[12].valid := 1, [1699].log_data[13].valid := 1, [1699].log_data[14].valid := 1, [1699].log_data[15].valid := 1, [1699].log_data[16].valid := 1, [1699].log_data[17].valid := 1, [1699].log_data[18].valid := 1, [1699].log_data[19].valid := 1, [1699].time.Year := 2023, [1699].time.Month := 1, [1699].time.Day := 15, [1699].time.Hour := 13, [1699].time.Minute := 59, [1699].time.Second := 59, [1700].log_data[0].min := 1.0, [1700].log_data[0].max := 1.0, [1700].log_data[0].total := 300.0, [1700].log_data[0].time := 300.0, [1700].log_data[0].valid := 1, [1700].log_data[1].valid := 1, [1700].log_data[2].valid := 1, [1700].log_data[3].valid := 1, [1700].log_data[4].valid := 1, [1700].log_data[5].valid := 1, [1700].log_data[6].valid := 1, [1700].log_data[7].valid := 1, [1700].log_data[8].valid := 1, [1700].log_data[9].valid := 1, [1700].log_data[10].valid := 1, [1700].log_data[11].valid := 1,
        [1700].log_data[12].valid := 1, [1700].log_data[13].valid := 1, [1700].log_data[14].valid := 1, [1700].log_data[15].valid := 1, [1700].log_data[16].valid := 1, [1700].log_data[17].valid := 1, [1700].log_data[18].valid := 1, [1700].log_data[19].valid := 1, [1700].time.Year := 2023, [1700].time.Month := 1, [1700].time.Day := 15, [1700].time.Hour := 14, [1700].time.Minute := 4, [1700].time.Second := 59, [1701].log_data[0].min := 1.0, [1701].log_data[0].max := 1.0, [1701].log_data[0].total := 300.0, [1701].log_data[0].time := 300.0, [1701].log_data[0].minminute := 5, [1701].log_data[0].maxminute := 5, [1701].log_data[0].valid := 1, [1701].log_data[1].valid := 1, [1701].log_data[2].valid := 1, [1701].log_data[3].valid := 1, [1701].log_data[4].valid := 1, [1701].log_data[5].valid := 1, [1701].log_data[6].valid := 1, [1701].log_data[7].valid := 1, [1701].log_data[8].valid := 1, [1701].log_data[9].valid := 1, [1701].log_data[10].valid := 1, [1701].log_data[11].valid := 1, [1701].log_data[12].valid := 1, [1701].log_data[13].valid := 1, [1701].log_data[14].valid := 1, [1701].log_data[15].valid := 1, [1701].log_data[16].valid := 1, [1701].log_data[17].valid := 1, [1701].log_data[18].valid := 1, [1701].log_data[19].valid := 1, [1701].time.Year := 2023, [1701].time.Month := 1, [1701].time.Day := 15, [1701].time.Hour := 14, [1701].time.Minute := 9, [1701].time.Second := 59, [1702].log_data[0].min := 1.0, [1702].log_data[0].max := 1.0, [1702].log_data[0].total := 300.0, [1702].log_data[0].time := 300.0, [1702].log_data[0].minminute := 10, [1702].log_data[0].maxminute := 10, [1702].log_data[0].valid := 1, [1702].log_data[1].valid := 1, [1702].log_data[2].valid := 1, [1702].log_data[3].valid := 1, [1702].log_data[4].valid := 1, [1702].log_data[5].valid := 1, [1702].log_data[6].valid := 1, [1702].log_data[7].valid := 1,
        [1702].log_data[8].valid := 1, [1702].log_data[9].valid := 1, [1702].log_data[10].valid := 1, [1702].log_data[11].valid := 1, [1702].log_data[12].valid := 1, [1702].log_data[13].valid := 1, [1702].log_data[14].valid := 1, [1702].log_data[15].valid := 1, [1702].log_data[16].valid := 1, [1702].log_data[17].valid := 1, [1702].log_data[18].valid := 1, [1702].log_data[19].valid := 1, [1702].time.Year := 2023, [1702].time.Month := 1, [1702].time.Day := 15, [1702].time.Hour := 14, [1702].time.Minute := 14, [1702].time.Second := 59, [1703].log_data[0].min := 1.0, [1703].log_data[0].max := 1.0, [1703].log_data[0].total := 300.0, [1703].log_data[0].time := 300.0, [1703].log_data[0].minminute := 15, [1703].log_data[0].maxminute := 15, [1703].log_data[0].valid := 1, [1703].log_data[1].valid := 1, [1703].log_data[2].valid := 1, [1703].log_data[3].valid := 1, [1703].log_data[4].valid := 1, [1703].log_data[5].valid := 1, [1703].log_data[6].valid := 1, [1703].log_data[7].valid := 1, [1703].log_data[8].valid := 1, [1703].log_data[9].valid := 1, [1703].log_data[10].valid := 1, [1703].log_data[11].valid := 1, [1703].log_data[12].valid := 1, [1703].log_data[13].valid := 1, [1703].log_data[14].valid := 1, [1703].log_data[15].valid := 1, [1703].log_data[16].valid := 1, [1703].log_data[17].valid := 1, [1703].log_data[18].valid := 1, [1703].log_data[19].valid := 1, [1703].time.Year := 2023, [1703].time.Month := 1, [1703].time.Day := 15, [1703].time.Hour := 14, [1703].time.Minute := 19, [1703].time.Second := 59, [1704].log_data[0].min := 1.0, [1704].log_data[0].max := 1.0, [1704].log_data[0].total := 300.0, [1704].log_data[0].time := 300.0, [1704].log_data[0].minminute := 20, [1704].log_data[0].maxminute := 20, [1704].log_data[0].valid := 1, [1704].log_data[1].valid := 1, [1704].log_data[2].valid := 1, [1704].log_data[3].valid := 1,
        [1704].log_data[4].valid := 1, [1704].log_data[5].valid := 1, [1704].log_data[6].valid := 1, [1704].log_data[7].valid := 1, [1704].log_data[8].valid := 1, [1704].log_data[9].valid := 1, [1704].log_data[10].valid := 1, [1704].log_data[11].valid := 1, [1704].log_data[12].valid := 1, [1704].log_data[13].valid := 1, [1704].log_data[14].valid := 1, [1704].log_data[15].valid := 1, [1704].log_data[16].valid := 1, [1704].log_data[17].valid := 1, [1704].log_data[18].valid := 1, [1704].log_data[19].valid := 1, [1704].time.Year := 2023, [1704].time.Month := 1, [1704].time.Day := 15, [1704].time.Hour := 14, [1704].time.Minute := 24, [1704].time.Second := 59, [1705].log_data[0].min := 1.0, [1705].log_data[0].max := 1.0, [1705].log_data[0].total := 300.0, [1705].log_data[0].time := 300.0, [1705].log_data[0].minminute := 25, [1705].log_data[0].maxminute := 25, [1705].log_data[0].valid := 1, [1705].log_data[1].valid := 1, [1705].log_data[2].valid := 1, [1705].log_data[3].valid := 1, [1705].log_data[4].valid := 1, [1705].log_data[5].valid := 1, [1705].log_data[6].valid := 1, [1705].log_data[7].valid := 1, [1705].log_data[8].valid := 1, [1705].log_data[9].valid := 1, [1705].log_data[10].valid := 1, [1705].log_data[11].valid := 1, [1705].log_data[12].valid := 1, [1705].log_data[13].valid := 1, [1705].log_data[14].valid := 1, [1705].log_data[15].valid := 1, [1705].log_data[16].valid := 1, [1705].log_data[17].valid := 1, [1705].log_data[18].valid := 1, [1705].log_data[19].valid := 1, [1705].time.Year := 2023, [1705].time.Month := 1, [1705].time.Day := 15, [1705].time.Hour := 14, [1705].time.Minute := 29, [1705].time.Second := 59, [1706].log_data[0].min := 1.0, [1706].log_data[0].max := 1.0, [1706].log_data[0].total := 300.0, [1706].log_data[0].time := 300.0, [1706].log_data[0].minminute := 30, [1706].log_data[0].maxminute := 30,
        [1706].log_data[0].valid := 1, [1706].log_data[1].valid := 1, [1706].log_data[2].valid := 1, [1706].log_data[3].valid := 1, [1706].log_data[4].valid := 1, [1706].log_data[5].valid := 1, [1706].log_data[6].valid := 1, [1706].log_data[7].valid := 1, [1706].log_data[8].valid := 1, [1706].log_data[9].valid := 1, [1706].log_data[10].valid := 1, [1706].log_data[11].valid := 1, [1706].log_data[12].valid := 1, [1706].log_data[13].valid := 1, [1706].log_data[14].valid := 1, [1706].log_data[15].valid := 1, [1706].log_data[16].valid := 1, [1706].log_data[17].valid := 1, [1706].log_data[18].valid := 1, [1706].log_data[19].valid := 1, [1706].time.Year := 2023, [1706].time.Month := 1, [1706].time.Day := 15, [1706].time.Hour := 14, [1706].time.Minute := 34, [1706].time.Second := 59, [1707].log_data[0].min := 1.0, [1707].log_data[0].max := 1.0, [1707].log_data[0].total := 300.0, [1707].log_data[0].time := 300.0, [1707].log_data[0].minminute := 35, [1707].log_data[0].maxminute := 35, [1707].log_data[0].valid := 1, [1707].log_data[1].valid := 1, [1707].log_data[2].valid := 1, [1707].log_data[3].valid := 1, [1707].log_data[4].valid := 1, [1707].log_data[5].valid := 1, [1707].log_data[6].valid := 1, [1707].log_data[7].valid := 1, [1707].log_data[8].valid := 1, [1707].log_data[9].valid := 1, [1707].log_data[10].valid := 1, [1707].log_data[11].valid := 1, [1707].log_data[12].valid := 1, [1707].log_data[13].valid := 1, [1707].log_data[14].valid := 1, [1707].log_data[15].valid := 1, [1707].log_data[16].valid := 1, [1707].log_data[17].valid := 1, [1707].log_data[18].valid := 1, [1707].log_data[19].valid := 1, [1707].time.Year := 2023, [1707].time.Month := 1, [1707].time.Day := 15, [1707].time.Hour := 14, [1707].time.Minute := 39, [1707].time.Second := 59, [1708].log_data[0].min := 1.0, [1708].log_data[0].max := 1.0,
